Universal Robots URScript: screwdriver.script

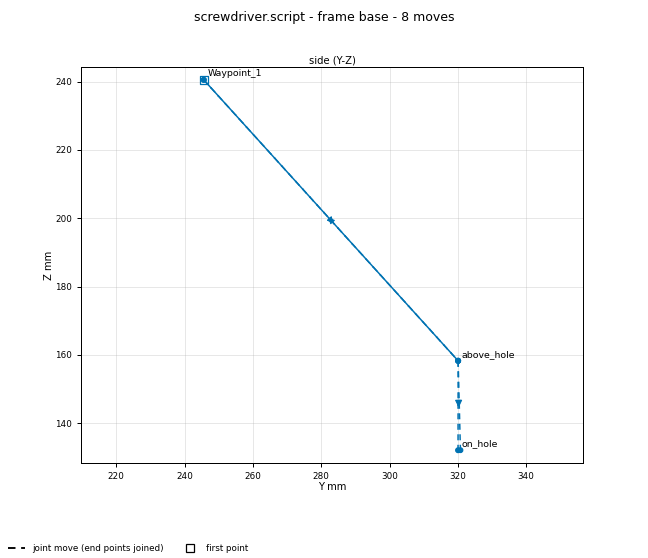
[picture p0: tool path of screwdriver.script in frame base, 8 of 54 moves have a stored position in this frame; points joined in program order, loops and branches not executed]
def unnamed():
  global _hidden_verificationVariable=0
  set_target_payload(1.710000, [0.052300, 0.000000, 0.046900], [0.000000, 0.000000, 0.000000, 0.000000, 0.000000, 0.000000])
  set_tool_communication(False, 115200, 0, 1, 1.5, 3.5)
  set_tool_output_mode(0)
  set_tool_digital_output_mode(0, 1)
  set_tool_digital_output_mode(1, 1)
  set_tool_voltage(0)
  set_gravity([0.0, 0.0, 9.82])
  set_safety_mode_transition_hardness(1)
  set_tcp(p[0.076,0.0,0.269,0.0,0.0,0.0])
  set_standard_analog_input_domain(0, 1)
  set_standard_analog_input_domain(1, 1)
  set_tool_analog_input_domain(0, 1)
  set_tool_analog_input_domain(1, 1)
  set_analog_outputdomain(0, 0)
  set_analog_outputdomain(1, 0)
  set_input_actions_to_default()
  global nb_vis_reusi=0
  global i_var_1=63
  global count_sec_touch=0
  global count_touch=0
  global erreur_vissage=0
  global perte_vis=0
  global count_vis=500
  global second_time_vis=0
  global rq_show_diag=0
  global count_pick_gig=5
  global count=495
  global should_i_vis=True
  # begin: URCap Installation Node
  #   Source: Robotiq_Screwdriving, 2.2.3.37910-alpha, Robotiq Inc.
  #   Type: Screwdriving
  #--------------------------------------------------------------------------------------------------
  # Screwdriver Constants
  #--------------------------------------------------------------------------------------------------
  RQ_REGULATION_MODE_CURRENT_WITH_RAMP_DOWN = 0
  RQ_REGULATION_MODE_ANGLE = 1
  RQ_REGULATION_MODE_TORQUE = 2
  RQ_REGULATION_MODE_SPEED = 3
  RQ_REGULATION_MODE_CURRENT = 4
  RQ_REGULATION_MODE_TIGHTENING = 5
  RQ_REGULATION_MODE_TORQUE_SPEED_CURRENT = 6
  RQ_ACTIVATE = True
  RQ_DIRECTION_CCW = False
  RQ_DIRECTION_CW = True
  RQ_MODE_NORMAL = False
  RQ_MODE_CALIBRATE = True
  RQ_SCREWDRIVER_ON = True
  RQ_SCREWDRIVER_OFF = False
  RQ_VACUUM_ON = True
  RQ_VACUUM_OFF = False
  RQ_MAX_SUPPLY_CURRENT_MA = 2000
  RQ_IN_ACTION = 0
  RQ_ANGLE_DETECTED = 1
  RQ_TORQUE_DETECTED = 2
  RQ_NO_DETECTION = 3
  RQ_SCREW_STATUS_ACTIVATION_IN_PROGRESS = 1
  RQ_SCREW_STATUS_ACTIVATION_DONE = 3
  RQ_SCREW_SUCCESS = 0
  RQ_SCREW_FAIL_ON_DISTANCE_MIN = 1
  RQ_SCREW_FAIL_ON_DISTANCE_MAX = 2
  RQ_SCREW_FAIL_ON_TIME_MAX = 3
  RQ_SCREW_FAIL_ON_SCREW_NOT_DETECTED = 4
  RQ_SCREW_FAIL_ON_SCREWDRIVER_NOT_ACTIVATED = 5
  RQ_SCREW_FAIL_ON_UNHANDLED_ERROR = 6
  RQ_SCREW_FAIL_ON_SCREWDRIVER_NOT_RESPONDING = 7
  RQ_SCREW_FAIL_ON_SCREWDRIVER_COMMUNICATION_LOST = 8
  RQ_SCREW_FAIL_ON_CONTACT_NOT_FOUND = 9
  RQ_SCREW_FAIL_WITHOUT_DETECTION = 10
  RQ_SCREW_SUCCESS_TEXT = "The screwdriving test is successful."
  RQ_SCREW_SUCCESS_TITLE_TEXT = "Screwdriving Test Success"
  RQ_PICK_SUCCESS = 0
  RQ_PICK_FAIL_ON_SCREW_NOT_READY = 1
  RQ_PICK_FAIL_ON_SCREW_NOT_DETECTED = 2
  RQ_PICK_FAIL_ON_FEEDER_NOT_READY = 3
  RQ_PICK_FAIL_ON_SCREWDRIVER_NOT_ACTIVATED = 5
  RQ_FEEDER_SCREW_PRESENT = 0
  RQ_PICK_SUCCESS_TEXT = "The pick test is successful."
  RQ_PICK_FAIL_ON_SCREW_NOT_READY_TEXT = "Screw not ready in feeder."
  RQ_PICK_FAIL_ON_SCREW_NOT_DETECTED_TEXT = "Screw not detected by screwdriver."
  RQ_PICK_FAIL_ON_FEEDER_NOT_READY_TEXT = "Feeder not ready."
  RQ_PICK_SUCCESS_TITLE_TEXT = "Pick Test Success"
  RQ_PICK_FAILED_TITLE_TEXT = "Pick Test Failed"
  RQ_SCREWDRIVER_NOT_ACTIVATED_TEXT = "Screwdriver is not activated. Please open Screwdriver Toolbar and click on Activate."
  RQ_MILLI_UNIT_TO_UNIT_FACTOR = 1000
  RQ_ENDLESS_TIMEOUT = 0
  RQ_UNUSED_PARAMETER = -1
  RQ_SCREW_FAIL_ON_DISTANCE_MIN_TEXT = "Minimum distance not reached."
  RQ_SCREW_FAIL_ON_DISTANCE_MAX_TEXT = "Maximum distance reached."
  RQ_SCREW_FAIL_ON_TIME_MAX_TEXT = "Maximum time reached."
  RQ_SCREW_FAIL_ON_NO_SCREW_TEXT = "No screw detected"
  RQ_SCREW_FAIL_TITLE = "Test Screw Failed"
  RQ_SCREW_FAIL_ON_UNHANDLED_ERROR_TEXT = "UE0 - Unhandled screw error"
  RQ_SCREW_FAIL_ON_SCREWDRIVER_NOT_RESPONDING_TEXT = "UE1 - Screwdriver not returning proper echo"
  RQ_SCREW_FAIL_ON_SCREWDRIVER_COMMUNICATION_LOST_TEXT = "UE2 - Screwdriver communication lost"
  RQ_SCREW_FAIL_ON_CONTACT_NOT_FOUND_TEXT = "UE3 - Contact with threads not found"
  RQ_SCREW_FAIL_WITHOUT_DETECTION_TEXT = "UE4 - Action finished without detection"
  RQ_TEACHING_OFF = 0
  RQ_TEACHING_ON = 1
  ###################################################
  #
  #  Fault types v2
  #
  ###################################################
  RQ_NO_FAULT = 0
  RQ_APPLICATION_WARNING = 1
  RQ_MOTOR_MINOR_ALARM = 2
  RQ_GENERAL_MINOR_ALARM = 4
  RQ_APPLICATION_MINOR_ALARM = 8
  RQ_MOTOR_MAJOR_ALARM = 16
  RQ_GENERAL_MAJOR_ALARM = 32
  RQ_APPLICATION_MAJOR_ALARM = 64
  RQ_CRITICAL_ALARM = 128

  RQ_NO_FAULT_MESSAGE = "NO_FAULT"
  RQ_APPLICATION_WARNING_MESSAGE = "APPLICATION_WARNING"
  RQ_MOTOR_MINOR_ALARM_MESSAGE = "MOTOR_MINOR_ALARM"
  RQ_GENERAL_MINOR_ALARM_MESSAGE = "GENERAL_MINOR_ALARM"
  RQ_APPLICATION_MINOR_ALARM_MESSAGE = "APPLICATION_MINOR_ALARM"
  RQ_MOTOR_MAJOR_ALARM_MESSAGE = "MOTOR_MAJOR_ALARM"
  RQ_GENERAL_MAJOR_ALARM_MESSAGE = "GENERAL_MAJOR_ALARM"
  RQ_APPLICATION_MAJOR_ALARM_MESSAGE = "APPLICATION_MAJOR_ALARM"
  RQ_CRITICAL_ALARM_MESSAGE = "CRITICAL_ALARM"

  ###################################################
  #
  #  Critical Alarm v2
  #
  ###################################################
  RQ_ACCELEROMETER_INIT = 1
  RQ_MOTOR_PWM_INIT = 2
  RQ_POSITION_SENSOR_INIT = 4
  RQ_GPIO_INIT = 8
  RQ_SOLENOID_INIT = 16
  RQ_FLASH_INIT = 32
  RQ_ADC_INIT = 64

  RQ_ACCELEROMETER_INIT_MESSAGE = "ACCELEROMETER_INIT"
  RQ_MOTOR_PWM_INIT_MESSAGE = "MOTOR_PWM_INIT"
  RQ_POSITION_SENSOR_INIT_MESSAGE = "POSITION_SENSOR_INIT"
  RQ_GPIO_INIT_MESSAGE = "GPIO_INIT"
  RQ_SOLENOID_INIT_MESSAGE = "SOLENOID_INIT"
  RQ_FLASH_INIT_MESSAGE = "FLASH_INIT"
  RQ_ADC_INIT_MESSAGE = "ADC_INIT"

  ###################################################
  #
  #  Application Warnings v2
  #
  ###################################################
  RQ_COMMUNICATION_NOT_READY = 1
  RQ_BLOCKED_AT_START = 2
  RQ_RESTRICTION_BEFORE_ANGLE = 4
  RQ_TIMEOUT = 8
  RQ_REG_WHILE_NOT_ACT = 16
  RQ_NOT_ACTIVATED = 32

  RQ_COMMUNICATION_NOT_READY_MESSAGE = "1 - COMMUNICATION_NOT_READY"
  RQ_BLOCKED_AT_START_MESSAGE = "2 - BLOCKED_AT_START"
  RQ_RESTRICTION_BEFORE_ANGLE_MESSAGE = "4 - RESTRICTION_BEFORE_ANGLE"
  RQ_TIMEOUT_MESSAGE = "8 - TIMEOUT"
  RQ_REGULATION_WHILE_NOT_ACT_MESSAGE = "16 - REGULATION_WHILE_NOT_ACT"
  RQ_NOT_ACTIVATED_MESSAGE = "32 - NOT_ACTIVATED"


  ###################################################
  #
  #  General Minor Alarm v2
  #
  ###################################################

  RQ_OVER_TEMPERATURE_SYSTEM = 2

  RQ_OVER_TEMPERATURE_SYSTEM_MESSAGE = "OVER_TEMPERATURE_SYSTEM"

  ###################################################
  #
  #  General Major Alarm v2
  #
  ###################################################

  RQ_E_STOP = 256
  RQ_OVER_CURRENT_SYSTEM = 512
  RQ_UNDER_VOLTAGE_24V = 1024
  RQ_UNDER_VOLTAGE_8V = 2048
  RQ_UNDER_VOLTAGE_3V = 4096

  RQ_E_STOP_MESSAGE = "E_STOP"
  RQ_OVER_CURRENT_SYSTEM_MESSAGE = "OVER_CURRENT_SYSTEM"
  RQ_UNDER_VOLTAGE_24V_MESSAGE = "UNDER_VOLTAGE_24V"
  RQ_UNDER_VOLTAGE_8V_MESSAGE = "UNDER_VOLTAGE_8V"
  RQ_UNDER_VOLTAGE_3V_MESSAGE = "UNDER_VOLTAGE_3V"

  ###################################################
  #
  #  Motor Minor Alarm v2
  #
  ###################################################
  RQ_CALIBRATION_PHASE_ERROR = 1
  RQ_CALIBRATION_POSITION_ERROR = 2
  RQ_CALIBRATION_PARAMETERS_ERROR = 4

  RQ_CALIBRATION_PHASE_ERROR_MESSAGE = "CALIBRATION_PHASE_ERROR"
  RQ_CALIBRATION_POSITION_ERROR_MESSAGE = "CALIBRATION_POSITION_ERROR"
  RQ_CALIBRATION_PARAMETERS_ERROR_MESSAGE = "CALIBRATION_PARAMETERS_ERROR"
  ###################################################
  #
  #  Motor Major Alarm v2
  #
  ###################################################
  RQ_UNDER_VOLTAGE = 1
  RQ_OVER_VOLTAGE = 2
  RQ_OVER_CURRENT_AC = 4
  RQ_OVER_CURRENT_DC = 8
  RQ_OVER_TEMP = 16
  RQ_POSITION_SENSOR_ERROR = 32
  RQ_PHASE_DRIVER_ERROR = 64
  RQ_PHASE_SENSOR_ERROR = 128

  RQ_UNDER_VOLTAGE_MESSAGE = "UNDER_VOLTAGE"
  RQ_OVER_VOLTAGE_MESSAGE = "OVER_VOLTAGE"
  RQ_OVER_CURRENT_AC_MESSAGE = "OVER_CURRENT_AC"
  RQ_OVER_CURRENT_DC_MESSAGE = "OVER_CURRENT_DC"
  RQ_OVER_TEMP_MESSAGE = "OVER_TEMP"
  RQ_POSITION_SENSOR_ERROR_MESSAGE = "POSITION_SENSOR_ERROR"
  RQ_PHASE_DRIVER_ERROR_MESSAGE = "PHASE_DRIVER_ERROR"
  RQ_PHASE_SENSOR_ERROR_MESSAGE = "PHASE_SENSOR_ERROR"
  global bash = rpc_factory("xmlrpc", "http://127.0.0.1:8000/bash")
  global logging_filename = str_cat("/tmp/screwing_info_",bash.date("+%Y_%m_%d_%H:%M:%S.csv"))
  #--------------------------------------------------------------------------------------------------
  #   Faults               2000[7-0]   Screwdriver fault types:
  #                                   0 = application warnings.[2501]
  #                                   1 = motor minor[2505]
  #                                   2 = general minor[2504]
  #                                   3 = application minor[2502]
  #                                   4 = motor major[2506]
  #                                   5 = general major[2504]
  #                                   6 = application major[2503]
  #                                   7 = critical[2500]
  #--------------------------------------------------------------------------------------------------
  def rq_get_screw_fault(slave_id=9):
    rq_error_list = [0,0,0,0,0,0,0,0]
    registers_200x = rq_comm_read_registers_200x(slave_id, RQ_READ_SCREWDRIVER_REGISTERS_SIZE)
    rq_error_type = registers_200x[0]

    if (rq_error_type == RQ_NO_FAULT):
      return rq_error_list
    end

    registers_250x = rq_comm_read_registers_250x(slave_id)
    rq_application_warnings = rq_extract_boolean_from_register_value(rq_error_type, 0)
    rq_motor_minor = rq_extract_boolean_from_register_value(rq_error_type, 1)
    rq_general_minor = rq_extract_boolean_from_register_value(rq_error_type, 2)
    rq_application_minor = rq_extract_boolean_from_register_value(rq_error_type, 3)
    rq_motor_major = rq_extract_boolean_from_register_value(rq_error_type, 4)
    rq_general_major = rq_extract_boolean_from_register_value(rq_error_type, 5)
    rq_application_major = rq_extract_boolean_from_register_value(rq_error_type, 6)
    rq_critical = rq_extract_boolean_from_register_value(rq_error_type, 7)

    if(rq_application_warnings):
     rq_error_list[0] = rq_extract_value_from_register_value(registers_250x[1], 0, 16)
    end
    if(rq_motor_minor):
     rq_error_list[1] = rq_extract_value_from_register_value(registers_250x[5], 0, 16)
    end
    if(rq_general_minor):
     rq_error_list[2] = rq_extract_value_from_register_value(registers_250x[4], 0, 8)
    end
    if(rq_application_minor):
     rq_error_list[3] = rq_extract_value_from_register_value(registers_250x[2], 0, 16)
    end
    if(rq_motor_major):
     rq_error_list[4] = rq_extract_value_from_register_value(registers_250x[6], 0, 16)
    end
    if(rq_general_major):
     rq_error_list[5] = rq_extract_value_from_register_value(registers_250x[4], 8, 16)
    end
    if(rq_application_major):
     rq_error_list[6] = rq_extract_value_from_register_value(registers_250x[3], 0, 16)
    end
    if(rq_critical):
     rq_error_list[7] = rq_extract_value_from_register_value(registers_250x[0], 0, 16)
    end

    return rq_error_list
  end

  #--------------------------------------------------------------------------------------------------
  #   Activate echo       2000[8]     Echo of the activate
  #--------------------------------------------------------------------------------------------------
  def rq_get_screw_activated_echo(slave_id=9):
      registers_200x = rq_comm_read_registers_200x(slave_id, RQ_READ_SCREWDRIVER_REGISTERS_SIZE)
      return rq_extract_is_screw_activated_echo(registers_200x)
  end
  def rq_extract_is_screw_activated_echo(registers_200x):
      return rq_extract_boolean_from_register_value(registers_200x[0], 8)
  end

  def rq_get_activation_and_screw_detection(slave_id):
    registers_200x = rq_comm_read_registers_200x(slave_id, RQ_READ_SCREWDRIVER_REGISTERS_SIZE)
    activation = rq_extract_is_screw_activated_echo(registers_200x)
    screw_detection = rq_extract_boolean_from_register_value(registers_200x[1], 12)

    return [activation, screw_detection]
  end
  #--------------------------------------------------------------------------------------------------
  #   Direction echo      2000[9]     Echo of the desired direction.
  #--------------------------------------------------------------------------------------------------
  def rq_get_screw_direction_echo(slave_id=9):
      registers_200x = rq_comm_read_registers_200x(slave_id, RQ_READ_SCREWDRIVER_REGISTERS_SIZE)
      return rq_extract_screw_direction_echo(registers_200x)
  end
  def rq_extract_screw_direction_echo(registers_200x):
      return rq_extract_boolean_from_register_value(registers_200x[0], 9)
  end

  #--------------------------------------------------------------------------------------------------
  #   Regulate echo       2000[11]    Echo of the regulate.
  #--------------------------------------------------------------------------------------------------
  def rq_get_screw_regulate_echo(slave_id=9):
      registers_200x = rq_comm_read_registers_200x(slave_id, RQ_READ_SCREWDRIVER_REGISTERS_SIZE)
      return rq_extract_screw_regulate_echo(registers_200x)
  end
  def rq_extract_screw_regulate_echo(registers_200x):
      return rq_extract_boolean_from_register_value(registers_200x[0], 11)
  end

  #--------------------------------------------------------------------------------------------------
  #   Screwdriver status  2000[13-12]     3 = Activation done
  #                                       1 = Activation in progress
  #                                       0 = Else
  #--------------------------------------------------------------------------------------------------
  def rq_get_screw_status(slave_id=9):
      registers_200x = rq_comm_read_registers_200x(slave_id, RQ_READ_SCREWDRIVER_REGISTERS_SIZE)
      return rq_extract_screw_status_echo(registers_200x)
  end
  def rq_extract_screw_status_echo(registers_200x):
      return rq_extract_value_from_register_value(registers_200x[0], 12, 2)
  end
  #--------------------------------------------------------------------------------------------------
  #   Action status       2000[15-14]     0 = initiating/doing an action
  #                                       1 = angle detected
  #                                       2 = torque detected
  #                                       3 = action finished without detection
  #--------------------------------------------------------------------------------------------------
  def rq_get_screw_action(slave_id=9):
      registers_200x = rq_comm_read_registers_200x(slave_id, RQ_READ_SCREWDRIVER_REGISTERS_SIZE)
      return rq_extract_value_from_register_value(registers_200x[0], 14, 2)
  end

  #--------------------------------------------------------------------------------------------------
  #   Regulation mode echo   2001[2-0]    0 = regulates speed, stops at desired current or timeout (ramp down at angle)
  #                                       1 = regulates speed, stops at desired current or timeout
  #                                       2 = regulates speed, stops at desired angle or timeout
  #                                       3 = regulates current, stops at timeout
  #                                       4 = regulates speed, stops at timeout
  #                                       5 = ?
  #                                       6 = regulate torque at stall (internal mode)
  #                                       7 = regultate torque (internal mode)
  #--------------------------------------------------------------------------------------------------
  def rq_get_screw_regulation_mode_echo(slave_id=9):
      registers_200x = rq_comm_read_registers_200x(slave_id, RQ_READ_SCREWDRIVER_REGISTERS_SIZE)
      return rq_extract_regulation_mode_echo(registers_200x)
  end
  def rq_extract_regulation_mode_echo(registers_200x):
      return rq_extract_value_from_register_value(registers_200x[1], 0, 2)
  end

  #--------------------------------------------------------------------------------------------------
  #   Vacuum screw detection 2001[12]     0 = not detected
  #                                       1 = detected
  #--------------------------------------------------------------------------------------------------
  def rq_is_screw_detected(slave_id=9):
      registers_200x = rq_comm_read_registers_200x(slave_id, RQ_READ_SCREWDRIVER_REGISTERS_SIZE)
      return rq_extract_boolean_from_register_value(registers_200x[1], 12)
  end

  #--------------------------------------------------------------------------------------------------
  #   Vacuum echo            2001[13]     0 = close
  #                                       1 = open
  #--------------------------------------------------------------------------------------------------
  def rq_get_screw_vacuum_echo(slave_id=9):
      registers_200x = rq_comm_read_registers_200x(slave_id, RQ_READ_SCREWDRIVER_REGISTERS_SIZE)
      return rq_extract_screw_vacuum_echo(registers_200x)
  end
  def rq_extract_screw_vacuum_echo(registers_200x):
      return rq_extract_boolean_from_register_value(registers_200x[1], 13)
  end

  #--------------------------------------------------------------------------------------------------
  #   Operation mode echo    2001[14]    Echo of the screwdriver mode
  #--------------------------------------------------------------------------------------------------
  def rq_get_screw_operation_mode_echo(slave_id=9):
      registers_200x = rq_comm_read_registers_200x(slave_id, RQ_READ_SCREWDRIVER_REGISTERS_SIZE)
      return rq_extract_screw_operation_mode(registers_200x)
  end
  def rq_extract_screw_operation_mode(registers_200x):
      return rq_extract_boolean_from_register_value(registers_200x[1], 14)
  end

  #--------------------------------------------------------------------------------------------------
  #   Rotation current echo   2002        Desired current to apply. 1 bit = 1 mA
  #--------------------------------------------------------------------------------------------------
  def rq_get_screw_rotation_current_echo_mA(slave_id=9):
      registers_200x = rq_comm_read_registers_200x(slave_id, RQ_READ_SCREWDRIVER_REGISTERS_SIZE)
      return rq_extract_rotation_current_echo(registers_200x)
  end
  def rq_extract_rotation_current_echo(registers_200x):
      return registers_200x[2]
  end

  #--------------------------------------------------------------------------------------------------
  #   Rotation speed echo     2003        Desired rotation speed to regulate in RPM
  #--------------------------------------------------------------------------------------------------
  def rq_get_screw_rotation_speed_echo_rpm(slave_id=9):
      registers_200x = rq_comm_read_registers_200x(slave_id, RQ_READ_SCREWDRIVER_REGISTERS_SIZE)
      return rq_extract_screw_rotation_speed_echo_rpm(registers_200x)
  end
  def rq_extract_screw_rotation_speed_echo_rpm(registers_200x):
      return registers_200x[3]
  end

  #--------------------------------------------------------------------------------------------------
  #   Actual delta angle      2004[15-0]-2005[15-8]    Actual delta angle in degrees
  #--------------------------------------------------------------------------------------------------
  def rq_get_screw_delta_angle_deg(slave_id=9):
      registers_200x = rq_comm_read_registers_200x(slave_id, RQ_READ_SCREWDRIVER_REGISTERS_SIZE)
      register_2005_8_15 = rq_extract_value_from_register_value(registers_200x[5], 8, 8)
      return registers_200x[4] + register_2005_8_15 * pow(2, 16)
  end

  #--------------------------------------------------------------------------------------------------
  #   Desired delta angle      2007[15-0]-2008[15-8]    Desired delta angle in degrees
  #--------------------------------------------------------------------------------------------------
  def rq_get_desired_delta_angle_deg(slave_id=9):
      registers_200x = rq_comm_read_registers_200x(slave_id, RQ_READ_SCREWDRIVER_REGISTERS_SIZE)
      register_2008_8_15 = rq_extract_value_from_register_value(registers_200x[8], 8, 8)
      return registers_200x[7] + register_2008_8_15 * pow(2, 16)
  end

  #--------------------------------------------------------------------------------------------------
  #   Actual current          2005[7-0]  Actual current, 1 bit = 100 mA
  #--------------------------------------------------------------------------------------------------
  def rq_get_screw_current_mA(slave_id=9):
      registers_200x = rq_comm_read_registers_200x(slave_id, RQ_READ_SCREWDRIVER_REGISTERS_SIZE)
      register_2005_0_7 = rq_extract_value_from_register_value(registers_200x[5], 0, 8)
      return register_2005_0_7 * 100
  end

  #--------------------------------------------------------------------------------------------------
  #   Actual rotation speed   2006    Actual rotation speed   RPM
  #--------------------------------------------------------------------------------------------------
  def rq_get_screw_rotation_speed_rpm(slave_id=9):
      registers_200x = rq_comm_read_registers_200x(slave_id, RQ_READ_SCREWDRIVER_REGISTERS_SIZE)
      return registers_200x[6]
  end

  #--------------------------------------------------------------------------------------------------
  #   Torque Threshold        2010
  #--------------------------------------------------------------------------------------------------
  def rq_get_torque_threshold_Nm(slave_id=9):
      registers_200x = rq_comm_read_registers_200x(slave_id, RQ_READ_SCREWDRIVER_REGISTERS_SIZE)
      return rq_extract_torque_threshold_echo(registers_200x) / 10000
  end
  def rq_extract_torque_threshold_echo(registers_200x):
      return rq_convert_unsigned16_to_signed16(registers_200x[10])
  end

  #--------------------------------------------------------------------------------------------------
  #   Torque Angle Slope      2011
  #--------------------------------------------------------------------------------------------------
  def rq_get_torque_slope(slave_id=9):
      registers_200x = rq_comm_read_registers_200x(slave_id, RQ_READ_SCREWDRIVER_REGISTERS_SIZE)
      return rq_extract_torque_angle_slope_echo(registers_200x)
  end
  def rq_extract_torque_angle_slope_echo(registers_200x):
      return rq_convert_unsigned16_to_signed16(registers_200x[11])
  end

  #--------------------------------------------------------------------------------------------------
  #   Torque Gain %     2012  value between 0 and 100. Default is 12
  #--------------------------------------------------------------------------------------------------
  def rq_get_torque_gain_pct(slave_id=9):
      registers = rq_read_registers(slave_id, 2012, 1, rq_xml_rpc_modbus_debug)
      return registers[0]
  end

  #--------------------------------------------------------------------------------------------------
  #   Debug register          6021
  #--------------------------------------------------------------------------------------------------
  def rq_get_screw_register_6021(slave_id=9):
      register_6020 = rq_comm_read_3_registers_6020(slave_id)

      return register_6020[1]
  end

  #--------------------------------------------------------------------------------------------------
  #   Debug register          6022
  #--------------------------------------------------------------------------------------------------
  def rq_get_screw_register_6022(slave_id=9):
      register_6020 = rq_comm_read_3_registers_6020(slave_id)

      return register_6020[2]
  end

  #--------------------------------------------------------------------------------------------------
  # Look for screwdriver activation
  #--------------------------------------------------------------------------------------------------
  def rq_screwdriver_is_activated(slave_id=9):
    registers_200x = rq_comm_read_registers_200x(slave_id, RQ_READ_SCREWDRIVER_REGISTERS_SIZE)

    return (rq_extract_screw_status_echo(registers_200x) == RQ_SCREW_STATUS_ACTIVATION_DONE) and rq_extract_is_screw_activated_echo(registers_200x)
  end

  #--------------------------------------------------------------------------------------------------
  # Returns True when all echo matches parameters
  #--------------------------------------------------------------------------------------------------
  def rq_screwdriver_echo_equal(slave_id, vacuum, rotation_current, regulate, direction, rotation_speed, operation_mode, regulation_mode, torque_threshold, torque_angle_slope):
    registers_200x = rq_comm_read_registers_200x(slave_id, RQ_READ_SCREWDRIVER_REGISTERS_SIZE)

    return (vacuum == rq_extract_screw_vacuum_echo(registers_200x)) and
           (rotation_current == rq_extract_rotation_current_echo(registers_200x)) and
           (regulate == rq_extract_screw_regulate_echo(registers_200x)) and
           (direction == rq_extract_screw_direction_echo(registers_200x)) and
           (rotation_speed == rq_extract_screw_rotation_speed_echo_rpm(registers_200x)) and
           (operation_mode == rq_extract_screw_operation_mode(registers_200x)) and
           (regulation_mode == rq_extract_regulation_mode_echo(registers_200x)) and
           (torque_threshold == rq_extract_torque_threshold_echo(registers_200x)) and
           (torque_angle_slope == rq_extract_torque_angle_slope_echo(registers_200x))

  end

  #--------------------------------------------------------------------------------------------------
  # Refresh registers 200x to get actual communication state. Return communication state.
  #--------------------------------------------------------------------------------------------------
  def rq_is_comm_lost(slave_id):
    rq_comm_read_registers_200x(slave_id, RQ_READ_SCREWDRIVER_REGISTERS_SIZE)

    return rq_comm_lost[rq_comm_slave_id_to_index(slave_id)]
  end

  #--------------------------------------------------------------------------------------------------
  # Returns the magnetic encoder count - Register 4000(LSB) - 4001(MSB)
  #--------------------------------------------------------------------------------------------------
  def rq_get_magnetic_encoder_count(slave_id=9):
      registers_lsb = rq_read_registers(slave_id, 4000, 1, rq_xml_rpc_modbus_debug)
      registers_msb = rq_read_registers(slave_id, 4001, 1, rq_xml_rpc_modbus_debug)

      return (registers_msb[0] * pow(2,16)) + registers_lsb[0]
  end

  #--------------------------------------------------------------------------------------------------
  # Returns the magnetic encoder error flag - Register 4002[15-13]
  #                                                         13 = Framing error
  #                                                         14 = Invalid command error
  #                                                         15 = Parity error
  #--------------------------------------------------------------------------------------------------
  def rq_get_magnetic_encoder_error_flag(slave_id=9):
      registers = rq_read_registers(slave_id, 4002, 1, rq_xml_rpc_modbus_debug)

      if (rq_extract_boolean_from_register_value(registers[0], 13)):
        return "Encoder error - Framing error"
      elif (rq_extract_boolean_from_register_value(registers[0], 14)):
        return "Encoder error - Invalid command error"
      elif (rq_extract_boolean_from_register_value(registers[0], 15)):
        return "Encoder error - Parity error"
      end

      return "No magnetic encoder error"
  end

  #--------------------------------------------------------------------------------------------------
  # Returns the magnetic encoder is ready - Register 4002[8]
  #--------------------------------------------------------------------------------------------------
  def rq_get_magnetic_encoder_ready(slave_id=9):
      registers = rq_read_registers(slave_id, 4002, 1,rq_xml_rpc_modbus_debug)

      return not rq_extract_boolean_from_register_value(registers[0], 8)
  end

  #--------------------------------------------------------------------------------------------------
  # Returns the magnetic encoder field strength - Register 4002[7-0]
  #--------------------------------------------------------------------------------------------------
  def rq_get_magnetic_encoder_field_strength(slave_id=9):
      registers = rq_read_registers(slave_id, 4002, 1, rq_xml_rpc_modbus_debug)

      return rq_extract_value_from_register_value(registers[0], 0, 8)
  end

  #--------------------------------------------------------------------------------------------------
  # Returns the CPU percent max live - Register 4003
  #--------------------------------------------------------------------------------------------------
  def rq_get_cpu_percent_max_live(slave_id=9):
      registers = rq_read_registers(slave_id, 4003, 1,rq_xml_rpc_modbus_debug)

      return registers[0]
  end

  #--------------------------------------------------------------------------------------------------
  # Returns the CPU percent max since boot - Register 4004
  #--------------------------------------------------------------------------------------------------
  def rq_get_cpu_percent_max_since_boot(slave_id=9):
      registers = rq_read_registers(slave_id, 4004, 1, rq_xml_rpc_modbus_debug)

      return registers[0]
  end

  #--------------------------------------------------------------------------------------------------
  # Returns the current motor analog Amps - Register 4005
  #--------------------------------------------------------------------------------------------------
  def rq_get_current_motor_amps(slave_id=9):
      registers = rq_read_registers(slave_id, 4005, 1, rq_xml_rpc_modbus_debug)

      return registers[0]/100
  end

  #--------------------------------------------------------------------------------------------------
  # Returns the analog 24v voltage - Register 4006
  #--------------------------------------------------------------------------------------------------
  def rq_get_analog_24_volt(slave_id=9):
      registers =rq_read_registers(slave_id, 4006, 1, rq_xml_rpc_modbus_debug)

      return registers[0]/100
  end

  #--------------------------------------------------------------------------------------------------
  # Returns the analog 8v8 voltage - Register 4007
  #--------------------------------------------------------------------------------------------------
  def rq_get_analog_8v8_volt(slave_id=9):
      registers = rq_read_registers(slave_id, 4007, 1, rq_xml_rpc_modbus_debug)

      return registers[0]/100
  end

  #--------------------------------------------------------------------------------------------------
  # Returns the microcontroller temperature Celsius - Register 4008
  #--------------------------------------------------------------------------------------------------
  def rq_get_uc_temp_celsius(slave_id=9):
      registers = rq_read_registers(slave_id, 4008, 1, rq_xml_rpc_modbus_debug)

      return registers[0]/100
  end

  #--------------------------------------------------------------------------------------------------
  # Returns the motor temperature Celsius - Register 4009
  #--------------------------------------------------------------------------------------------------
  def rq_get_motor_temp_celsius(slave_id=9):
      registers = rq_read_registers(slave_id, 4009, 1,rq_xml_rpc_modbus_debug)

      return registers[0]/100
  end

  #--------------------------------------------------------------------------------------------------
  # Returns the vacuum pressure Psi - Register 4010
  #--------------------------------------------------------------------------------------------------
  def rq_get_vacuum_pressure_kpa(slave_id=9):
      registers = rq_read_registers(slave_id, 4010, 1, rq_xml_rpc_modbus_debug)

      return rq_convert_unsigned16_to_signed16(registers[0]) / 100
  end

  #--------------------------------------------------------------------------------------------------
  # Returns the estimated load torque - Register 4012
  #--------------------------------------------------------------------------------------------------
  def rq_get_load_nm(slave_id=9):
      registers = rq_read_registers(slave_id, 4012, 1, rq_xml_rpc_modbus_debug)

      return registers[0]/1000
  end

  #--------------------------------------------------------------------------------------------------
  # Returns the estimated maximum load torque - Register 4013
  #--------------------------------------------------------------------------------------------------
  def rq_get_max_load_nm(slave_id=9):
      registers = rq_read_registers(slave_id, 4013, 1, rq_xml_rpc_modbus_debug)

      return registers[0]/1000
  end

  #--------------------------------------------------------------------------------------------------
  # add all diagnostic registers output in Polyscope Log tab.
  #--------------------------------------------------------------------------------------------------
  def rq_log_screw_diag_registers(slave_id=9):
    textmsg("magnetic encoder count : ", rq_get_magnetic_encoder_count(slave_id))
    textmsg("magnetic encoder is ready : ", rq_get_magnetic_encoder_ready(slave_id))
    textmsg("magnetic encoder error flag : ", rq_get_magnetic_encoder_error_flag(slave_id))
    textmsg("magnetic encoder field strength : ", rq_get_magnetic_encoder_field_strength(slave_id))
    textmsg("CPU percent max LIVE : ", rq_get_cpu_percent_max_live(slave_id))
    textmsg("CPU percent max since boot : ", rq_get_cpu_percent_max_since_boot(slave_id))
    textmsg("current motor analog Amps : ", rq_get_current_motor_amps(slave_id))
    textmsg("analog 24v voltage : ", rq_get_analog_24_volt(slave_id))
    textmsg("analog 8v8 voltage : ", rq_get_analog_8v8_volt(slave_id))
    textmsg("microcontroller temp Celsius : ", rq_get_uc_temp_celsius(slave_id))
    textmsg("motor temp Celsius : ", rq_get_motor_temp_celsius(slave_id))
    textmsg("vacuum pressure Kpa : ", rq_get_vacuum_pressure_kpa(slave_id))
    textmsg("estimated load torque Nm LIVE : ", rq_get_load_nm(slave_id))
    textmsg("estimated maximum load torque Nm :", rq_get_max_load_nm(slave_id))
  end

  #--------------------------------------------------------------------------------------------------
  #   Pressure sensor offset        441 (100bit = kPa (signed))
  #                                 pressure_offset in kpa
  #
  #--------------------------------------------------------------------------------------------------
  def get_pressure_sensor_offset(slave_id = 9):
    registers = rq_read_registers(slave_id, 441, 1, rq_xml_rpc_modbus_debug)

    return rq_convert_unsigned16_to_signed16(registers[0]) / 100
  end

  #--------------------------------------------------------------------------------------------------
  # Convert unsigned 16 bits integer to signed 16 bits integer
  #--------------------------------------------------------------------------------------------------
  def rq_convert_unsigned16_to_signed16(value):
    if (value >= 32768):
      return value - 65536
    end
    return value
  end
  #--------------------------------------------------------------------------------------------------
  #   Register            1000        Action request
  #
  #   Regulation mode     1000[2-0]   0 = regulates speed, stops at desired current or timeout
  #                                   1 = regulates speed, with ramp down, stops at desired angle or timeout
  #                                   2-7 = unused
  #   Activate            1000[8]     0 = Resetting errors
  #                                   1 = Allows the screwdriver to do an action
  #   Rotation direction  1000[9]     0 = Clockwise (screwing)
  #                                   1 = Counter-clockwise (unscrewing)
  #   Regulate            1000[11]    0 = doing nothing (stop movement)
  #                                   1 = regulating movement
  #   Teaching            1000[12]    0 = inactive
  #                                   1 = active
  #   Vacuum activation   1000[13]    0 = close
  #                                   1 = open
  #   Operation mode      1000[14]    0 = normal mode (Torque mode)
  #                                   1 = calibration mode (Current Mode)
  #   Command modify      1000[15]    0 = new command
  #                                   1 = modify command
  #--------------------------------------------------------------------------------------------------
  #   Register            1001[15-0]  Max supply current
  #                                   Range 0-65535 (1 bit = 1 mA)
  #--------------------------------------------------------------------------------------------------
  #   Register            1002[15-0]   Desired rotation current
  #                                    Range 0-65535 (1 bit = 1 mA)
  #--------------------------------------------------------------------------------------------------
  #   Register            1003        Desired rotation speed in RPM
  #                                   Range 16bit = 65Krpm
  #--------------------------------------------------------------------------------------------------
  #   Register            1004[15-0]-1005[15-8]   Desired rotation delta angle
  #                                               Desired delta angle to attain
  #                                               24bit = 46 kdegrees
  #--------------------------------------------------------------------------------------------------
  #   Register            1005[7-0]   Rotation timeout
  #                                   Timeout of regulated movement (8bit = 25.5s), 1bit = 0.1s
  #--------------------------------------------------------------------------------------------------
  #   Register            1006        Torque Threshold
  #
  #--------------------------------------------------------------------------------------------------
  #   Register            1007        Torque Angle Slope
  #
  #--------------------------------------------------------------------------------------------------
  def rq_set_screw_registers_100x(slave_id, regulation_mode, activate, direction, operation_mode, regulate, teaching,
  vacuum, rotation_current, max_supply_current_mA, rotation_speed_rpm, rotation_delta_angle, rotation_timeout_ms,
  torque_threshold, torque_angle_slope, modify_command = False):
      registers_100x = [0, 0, 0, 0, 0, 0, 0, 0]
      registers_100x[0] = rq_insert_value_in_register_value(registers_100x[0], 0, 3, regulation_mode)
      registers_100x[0] = rq_insert_boolean_in_register_value(registers_100x[0], 8, activate)
      registers_100x[0] = rq_insert_boolean_in_register_value(registers_100x[0], 9, direction)
      registers_100x[0] = rq_insert_boolean_in_register_value(registers_100x[0], 11, regulate)
      registers_100x[0] = rq_insert_value_in_register_value(registers_100x[0], 12, 1, teaching)
      registers_100x[0] = rq_insert_boolean_in_register_value(registers_100x[0], 13, vacuum)
      registers_100x[0] = rq_insert_boolean_in_register_value(registers_100x[0], 14, operation_mode)
      registers_100x[0] = rq_insert_boolean_in_register_value(registers_100x[0], 15, modify_command)

      registers_100x[1] = max_supply_current_mA

      registers_100x[2] = rotation_current

      registers_100x[3] = rotation_speed_rpm

      rotation_angle_lsb = floor(rotation_delta_angle % pow(2, 16))
      rotation_angle_msb = floor((rotation_delta_angle -  rotation_angle_lsb) / pow(2, 16))

      registers_100x[4] = rotation_angle_lsb
      registers_100x[5] = rq_insert_msb_in_register_value(registers_100x[5], rotation_angle_msb)
      registers_100x[5] = rq_insert_lsb_in_register_value(registers_100x[5], floor(rotation_timeout_ms / 100))

      registers_100x[6] = torque_threshold
      registers_100x[7] = torque_angle_slope

      rq_comm_write_registers_100x(slave_id, registers_100x, 8)
  end

  #--------------------------------------------------------------------------------------------------
  #   Activate screwdriver, sequence:
  #   1 - Reset screwdriver (activate = False) and wait echo
  #   2 - Activate screwdriver (activate = True) and wait echo and status
  #--------------------------------------------------------------------------------------------------
  def rq_screw_activate(slave_id = 9):
      while(rq_get_screw_activated_echo(slave_id)):
          registers_100x = rq_comm_get_registers_100x(slave_id, 8)
          registers_100x[0] = rq_insert_boolean_in_register_value(registers_100x[0], 8, False)
          rq_comm_write_registers_100x(slave_id, registers_100x, 8)
          sleep(0.1)
      end

      while(not rq_get_screw_activated_echo(slave_id) or rq_get_screw_status(slave_id) != RQ_SCREW_STATUS_ACTIVATION_DONE):
          registers_100x = rq_comm_get_registers_100x(slave_id, 8)
          registers_100x[0] = rq_insert_boolean_in_register_value(registers_100x[0], 8, True)
          rq_comm_write_registers_100x(slave_id, registers_100x, 8)
          sleep(0.1)
      end
  end

  #--------------------------------------------------------------------------------------------------
  #   Regulate            1000[11]    0 = doing nothing (stop movement)
  #                                   1 = regulating movement
  #--------------------------------------------------------------------------------------------------
  def rq_set_screw_regulate(slave_id, regulate):
      registers_100x = rq_comm_get_registers_100x(slave_id, 8)
      registers_100x[0] = rq_insert_boolean_in_register_value(registers_100x[0], 11, regulate)
      rq_comm_write_registers_100x(slave_id, registers_100x, 8)
  end

  #--------------------------------------------------------------------------------------------------
  #   Torque gain %            1008   torque gain is a value between 0 and 100. The default value is 12.
  #
  #--------------------------------------------------------------------------------------------------
  def rq_set_torque_gain_pct(torque_gain = 12, slave_id=9):
    rq_write_registers(slave_id, 1008, [torque_gain], rq_xml_rpc_modbus_debug)
  end

  #--------------------------------------------------------------------------------------------------
  #   Vacuum command on
  #--------------------------------------------------------------------------------------------------
  def rq_screw_vacuum_on(slave_id = 9):
      rq_set_screw_vacuum(True, slave_id)
  end

  #--------------------------------------------------------------------------------------------------
  #   Vacuum command off
  #--------------------------------------------------------------------------------------------------
  def rq_screw_vacuum_off(slave_id = 9):
      rq_set_screw_vacuum(False, slave_id)
  end

  #--------------------------------------------------------------------------------------------------
  #   Vacuum command off and regulate to false
  #--------------------------------------------------------------------------------------------------

  def rq_screw_vacuum_off_and_stop_regulate(slave_id=9):
    registers_100x = rq_comm_get_registers_100x(slave_id, 8)
    registers_200x = rq_comm_read_registers_200x(slave_id, RQ_READ_SCREWDRIVER_REGISTERS_SIZE)

    activate = rq_extract_boolean_from_register_value(registers_200x[0], 8)
    rotation_direction = rq_extract_boolean_from_register_value(registers_200x[0], 9)
    regulation_mode = rq_extract_value_from_register_value(registers_200x[1], 0, 2)
    operation_mode = rq_extract_value_from_register_value(registers_200x[1], 14, 1)
    regulate = False
    vacuum = False

    registers_100x[0] = rq_insert_value_in_register_value(registers_100x[0], 0, 2, regulation_mode)
    registers_100x[0] = rq_insert_boolean_in_register_value(registers_100x[0], 8, activate)
    registers_100x[0] = rq_insert_boolean_in_register_value(registers_100x[0], 9, rotation_direction)
    registers_100x[0] = rq_insert_boolean_in_register_value(registers_100x[0], 11, regulate)
    registers_100x[0] = rq_insert_boolean_in_register_value(registers_100x[0], 13, vacuum)
    registers_100x[0] = rq_insert_value_in_register_value(registers_100x[0], 14, 2, operation_mode)

    rq_comm_write_registers_100x(slave_id, registers_100x, 8)
  end

  #--------------------------------------------------------------------------------------------------
  #   Vacuum command         1000[13]     0 = close
  #                                       1 = open
  #--------------------------------------------------------------------------------------------------
  def rq_set_screw_vacuum(vacuum, slave_id = 9):
    registers_100x = rq_comm_get_registers_100x(slave_id, 8)
    registers_200x = rq_comm_read_registers_200x(slave_id, RQ_READ_SCREWDRIVER_REGISTERS_SIZE)

    activate = rq_extract_boolean_from_register_value(registers_200x[0], 8)
    rotation_direction = rq_extract_boolean_from_register_value(registers_200x[0], 9)
    regulate = rq_extract_boolean_from_register_value(registers_200x[0], 11)
    regulation_mode = rq_extract_value_from_register_value(registers_200x[1], 0, 2)
    operation_mode = rq_extract_value_from_register_value(registers_200x[1], 14, 1)

    registers_100x[0] = rq_insert_value_in_register_value(registers_100x[0], 0, 2, regulation_mode)
    registers_100x[0] = rq_insert_boolean_in_register_value(registers_100x[0], 8, activate)
    registers_100x[0] = rq_insert_boolean_in_register_value(registers_100x[0], 9, rotation_direction)
    registers_100x[0] = rq_insert_boolean_in_register_value(registers_100x[0], 11, regulate)
    registers_100x[0] = rq_insert_boolean_in_register_value(registers_100x[0], 13, vacuum)
    registers_100x[0] = rq_insert_value_in_register_value(registers_100x[0], 14, 2, operation_mode)

    rq_comm_write_registers_100x(slave_id, registers_100x, 8)
  end

  #--------------------------------------------------------------------------------------------------
  #   Set Pressure sensor offset        441 (100bit = kPa (signed))
  #                                      pressure_offset in kpa
  #
  #--------------------------------------------------------------------------------------------------
  def set_pressure_sensor_offset(pressure_offset=0, slave_id = 9):
    SAVE_PRESSURE_OFFSET = 56
    KPA_TO_BIT = 100

    offset_in_bit = rq_convert_unsigned32_to_signed16(pressure_offset * KPA_TO_BIT)
    rq_write_registers(slave_id, 441, [offset_in_bit], rq_xml_rpc_modbus_debug)

    save_pressure_offset_msb = floor(SAVE_PRESSURE_OFFSET * pow(2,8))
    rq_write_registers(slave_id, 440, [save_pressure_offset_msb], rq_xml_rpc_modbus_debug)
  end

  #--------------------------------------------------------------------------------------------------
  # Convert unsigned 32 bits integer to signed 16 bits integer
  #--------------------------------------------------------------------------------------------------
  def rq_convert_unsigned32_to_signed16(value):
    if (value < 0):
      return value + 65536
    end
    return value
  end

  #--------------------------------------------------------------------------------------------------
  #   Reset Pressure sensor offset to ambient pressure       440
  #
  #--------------------------------------------------------------------------------------------------
  def reset_pressure_sensor_offset(slave_id = 9):
    RESET_PRESSURE_OFFSET = 131

    reset_pressure_offset_msb = floor(RESET_PRESSURE_OFFSET * pow(2,8))
    rq_write_registers(slave_id, 440, [reset_pressure_offset_msb], rq_xml_rpc_modbus_debug)
  end
  global rq_feeder_timeout = 90
  global rq_pick_rotation_speed = 200

  def rq_is_feeder_screw_ready(ready_input):
    return get_standard_digital_in(ready_input)
  end

  def rq_is_feeder_status_ok(feeder_status):
    return get_standard_digital_in(feeder_status)
  end

  def rq_wait_for_feeder_status_ok(feeder_status, timeout):
    time_step = 0.008

    if(not rq_is_feeder_status_ok(feeder_status)):
      textmsg("Waiting for feeder status.")
    end

    while((not rq_is_feeder_status_ok(feeder_status)) and (timeout > 0)):
          sleep(time_step)
          timeout = timeout - time_step
    end

    return rq_is_feeder_status_ok(feeder_status)
  end

  def rq_pick_screw(screw_pose, status_input, ready_input, test_in_action=False, approach_dist=10, rotation_speed=rq_pick_rotation_speed,
  pick_speed=25, timeout=rq_feeder_timeout, retract_speed=40, direction=RQ_DIRECTION_CCW, slave_id=9):
      global thread_slave_id = slave_id
      global thread_rotation_speed = rotation_speed
      global thread_direction = direction

      rq_screwdriver_index = rq_comm_slave_id_to_index(slave_id)
      approach_dist_m = norm(approach_dist) / 1000
      pick_speed_m = pick_speed / 1000
      retract_speed_m = retract_speed / 1000
      approach_in_screw_frame = p[0, 0, -approach_dist_m, 0, 0, 0]

      def move_to_approach(screw_pose_in_base_frame, approach_in_screw_frame, blend=True):
        approach_in_base_frame = pose_trans(screw_pose_in_base_frame, approach_in_screw_frame)
        dist_to_approach = point_dist(get_actual_tcp_pose(), approach_in_base_frame)
        offset = 0.005
        blend_radius = offset * 0.99
        if blend and (dist_to_approach > blend_radius):
          approach_to_blend_in_base_frame = pose_trans(approach_in_base_frame, p[0, 0, -offset, 0, 0, 0])
          movel(approach_to_blend_in_base_frame, r=blend_radius)
        else:
          movel(approach_in_base_frame)
        end
      end

      def move_to_retract_servoj(ready_input, robot_speed, slave_id):
        max_distance = 0.05
        linear_speed = -robot_speed
        time_step = 0.008
        initial_pose = get_actual_tcp_pose()
        linear_step = linear_speed * time_step
        distance = 0

        while(get_standard_digital_in(ready_input)):
          distance = distance + linear_step
          next_pose = pose_trans(initial_pose, p[0, 0, distance, 0, 0, 0])
          next_joint_position = get_inverse_kin(next_pose)
          servoj(next_joint_position, t=time_step)

          if (norm(distance) >= max_distance):
            break
          end
        end
        stopj(2)
      end

      def move_to_screw(screw_pose_in_base_frame, robot_speed):
          movel(screw_pose_in_base_frame, v = robot_speed)
      end

      thread start_screwdriver_thread():
        torque_Nm = 1
        rotation_current_mA = floor(torque_Nm * 100)
        rotation_delta_angle = 100
        rotation_timeout_ms = 0
        torque_threshold = 0
        torque_angle_slope = 0
        retries = 40

        rq_set_screw_registers_100x(thread_slave_id, RQ_REGULATION_MODE_SPEED, RQ_ACTIVATE, thread_direction,
        RQ_MODE_NORMAL, RQ_SCREWDRIVER_ON, RQ_TEACHING_OFF, RQ_VACUUM_ON, rotation_current_mA, RQ_MAX_SUPPLY_CURRENT_MA,
        thread_rotation_speed, rotation_delta_angle, rotation_timeout_ms, torque_threshold, torque_angle_slope)

        while (not rq_screwdriver_echo_equal(thread_slave_id, RQ_VACUUM_ON, rotation_current_mA, RQ_SCREWDRIVER_ON,
        thread_direction, thread_rotation_speed, RQ_MODE_NORMAL, RQ_REGULATION_MODE_SPEED, torque_threshold, torque_angle_slope)):
          if ((retries <= 0) or (rq_comm_lost[rq_comm_slave_id_to_index(thread_slave_id)])):
            break
          end
          sleep(0.008)
          rq_set_screw_registers_100x(thread_slave_id, RQ_REGULATION_MODE_SPEED, RQ_ACTIVATE, thread_direction,
          RQ_MODE_NORMAL, RQ_SCREWDRIVER_ON, RQ_TEACHING_OFF, RQ_VACUUM_ON, rotation_current_mA, RQ_MAX_SUPPLY_CURRENT_MA,
           thread_rotation_speed, rotation_delta_angle, rotation_timeout_ms, torque_threshold, torque_angle_slope)
          retries = retries - 1
        end
      end

      def stop_screwdriver(slave_id = 9):
          rotation_current_mA = 0
          rotation_delta_angle = 100
          rotation_timeout_ms = 0
          rotation_speed_rpm = 0
          torque_threshold = 0
          torque_angle_slope = 0

          rq_set_screw_registers_100x(slave_id, RQ_REGULATION_MODE_SPEED, RQ_ACTIVATE, RQ_DIRECTION_CW, RQ_MODE_NORMAL,
          RQ_SCREWDRIVER_OFF, RQ_TEACHING_OFF, RQ_VACUUM_ON, rotation_current_mA, RQ_MAX_SUPPLY_CURRENT_MA,
          rotation_speed_rpm, rotation_delta_angle, rotation_timeout_ms, torque_threshold, torque_angle_slope)

          while (RQ_SCREWDRIVER_ON == rq_get_screw_regulate_echo(slave_id)):
            if(rq_comm_lost[rq_comm_slave_id_to_index(slave_id)]):
              break
            end
            sleep(0.008)
            rq_set_screw_registers_100x(slave_id, RQ_REGULATION_MODE_SPEED, RQ_ACTIVATE, RQ_DIRECTION_CW, RQ_MODE_NORMAL,
            RQ_SCREWDRIVER_OFF,  RQ_TEACHING_OFF, RQ_VACUUM_ON, rotation_current_mA, RQ_MAX_SUPPLY_CURRENT_MA,
            rotation_speed_rpm, rotation_delta_angle, rotation_timeout_ms, torque_threshold, torque_angle_slope)
          end
      end

      def wait_for_screw_present(status_input, ready_input, timeout):
        time_step = 1
        screw_ready = get_standard_digital_in(ready_input)

        while(not screw_ready):
          if (timeout <= 0):
            feeder_status = get_standard_digital_in(status_input)
            if (not feeder_status):
              return RQ_PICK_FAIL_ON_FEEDER_NOT_READY
            end
            return RQ_PICK_FAIL_ON_SCREW_NOT_READY
          end
          sleep(time_step)
          timeout = timeout - time_step
          screw_ready = get_standard_digital_in(ready_input)
        end

        return RQ_FEEDER_SCREW_PRESENT
      end

      thread stop_vacuum_thread():
        rq_set_screw_vacuum(False, thread_slave_id)
         while (RQ_VACUUM_ON == rq_get_screw_vacuum_echo(thread_slave_id)):
           if(rq_comm_lost[rq_comm_slave_id_to_index(thread_slave_id)]):
             break
           end
           sleep(0.008)
           rq_set_screw_vacuum(False, thread_slave_id)
         end
      end

      thread screw_detection():
        global screw_detected_flag = False
        index = rq_comm_slave_id_to_index(thread_slave_id)
        while (not rq_is_screw_detected(thread_slave_id)):
          if(rq_comm_lost[index]):
            break
          end
          global screw_detected_flag = False
          sleep(0.008)
        end
        global screw_detected_flag = not rq_comm_lost[index]
      end

      def start_screw_detection():
        global screw_detected_flag = False
        return run screw_detection()
      end

      def screw_detected():
        return screw_detected_flag
      end

      def wait_for_screw_detected(timeout):
        time_step = 0.1
        detected = False
        thread_id = start_screw_detection()
        while (timeout >= 0):
          sleep(time_step)
          timeout = timeout - time_step
          if (screw_detected()):
            detected = True
            break
          end
        end
        kill thread_id
        return detected
      end

      thread peck():
        while (True):
          movel(pose_trans(get_target_tcp_pose(), p[0, 0, -0.004, 0, 0, 0]), a=0.15, v=0.25)
          movel(pose_trans(get_target_tcp_pose(), p[0, 0, 0.004, 0, 0, 0]), a=0.15, v=0.25)
        end
      end

    #--------------------------------------------------------------------------------------------------
    # Process begins here
    #--------------------------------------------------------------------------------------------------
      if ((not test_in_action) and (rq_wait_for_feeder_status_ok(status_input, timeout))):
        stop_vacuum_thread_id = run stop_vacuum_thread()
        move_to_approach(screw_pose, approach_in_screw_frame)
        join stop_vacuum_thread_id
        if (rq_comm_lost[rq_screwdriver_index]):
          textmsg(RQ_SCREW_FAIL_ON_SCREWDRIVER_COMMUNICATION_LOST_TEXT)

          return RQ_SCREW_FAIL_ON_SCREWDRIVER_COMMUNICATION_LOST
        end
      elif(not rq_is_feeder_status_ok(status_input)):
        sleep(0.008)
        return RQ_PICK_FAIL_ON_FEEDER_NOT_READY
      end

      if ((not rq_is_feeder_screw_ready(ready_input)) and (rq_wait_for_feeder_status_ok(status_input, timeout))):
        move_to_approach(screw_pose, approach_in_screw_frame, blend=False)
      elif(not rq_is_feeder_status_ok(status_input)):
        return RQ_PICK_FAIL_ON_FEEDER_NOT_READY
      end

      feeder_result = wait_for_screw_present(status_input, ready_input, timeout)
      if (RQ_FEEDER_SCREW_PRESENT != feeder_result):
          return feeder_result
      end

      start_screwdriver_thread_id = run start_screwdriver_thread()
      move_to_screw(screw_pose, pick_speed_m)
      join start_screwdriver_thread_id

      if (rq_comm_lost[rq_screwdriver_index]):
        textmsg(RQ_SCREW_FAIL_ON_SCREWDRIVER_COMMUNICATION_LOST_TEXT)
        kill start_screwdriver_thread_id

        return RQ_SCREW_FAIL_ON_SCREWDRIVER_COMMUNICATION_LOST
      end

      if (not rq_screwdriver_is_activated(slave_id)):
        return RQ_PICK_FAIL_ON_SCREWDRIVER_NOT_ACTIVATED
      end

      peck_thread_id = run peck()
      wait_for_screw_detected(2)
      kill peck_thread_id
      move_to_retract_servoj(ready_input, retract_speed_m, slave_id)
      is_screw_detected = wait_for_screw_detected(2)
      stop_screwdriver(slave_id)

      if (rq_comm_lost[rq_screwdriver_index]):
        textmsg(RQ_SCREW_FAIL_ON_SCREWDRIVER_COMMUNICATION_LOST_TEXT)

        return RQ_SCREW_FAIL_ON_SCREWDRIVER_COMMUNICATION_LOST
      end
      if (not is_screw_detected):
          return RQ_PICK_FAIL_ON_SCREW_NOT_DETECTED
      end

      return RQ_PICK_SUCCESS
  end
  global rq_screwdriver_faults = [0,0,0,0,0,0,0,0]
  global rq_max_thread_contact_distance = 0.05
  global rq_unhandled_error = RQ_NO_FAULT
  global rq_fs_speed = 0.008
  global rq_log_screwing = False
  copilot_kinematics_rpc_server = rpc_factory("xmlrpc","http://localhost:4251/")
  global app_time = 0
  global rq_find_surface_time = 0
  global rq_screwing_time = 0

  thread app_timer():
    step_time = get_steptime()
    app_time = 0
    while(True):
      app_time = app_time + step_time
      sleep(step_time)
    end
  end

  def rq_screw(operation_mode, regulation_mode, rotation_current, rotation_speed, rotation_angle, timeout, teaching,
  torque_threshold, torque_angle_slope, direction=RQ_DIRECTION_CW, slave_id=9):
    direction = direction
    activation = RQ_ACTIVATE
    regulate = RQ_SCREWDRIVER_ON
    vacuum = rq_get_screw_vacuum_echo(slave_id)
    rotation_speed_raw = rotation_speed
    max_supply_current = RQ_MAX_SUPPLY_CURRENT_MA
    time_max = timeout * 1000
    index = rq_comm_slave_id_to_index(slave_id)

    if(timeout == RQ_UNUSED_PARAMETER):
      time_max = RQ_ENDLESS_TIMEOUT
    end

    retries = 40
    rq_set_screw_registers_100x(slave_id, regulation_mode, activation, direction, operation_mode, regulate, teaching, vacuum,
                                rotation_current, max_supply_current, rotation_speed_raw, rotation_angle, time_max,
                                torque_threshold, torque_angle_slope)
    while (not rq_screwdriver_echo_equal(slave_id, vacuum, rotation_current, regulate, direction, rotation_speed_raw, operation_mode, regulation_mode, torque_threshold, torque_angle_slope)):
      if ((retries <= 0) or (rq_comm_lost[index])):
        return False
      end
      sleep(0.008)
      rq_set_screw_registers_100x(slave_id, regulation_mode, activation, direction, operation_mode, regulate, teaching, vacuum,
                                  rotation_current, max_supply_current, rotation_speed_raw, rotation_angle, time_max,
                                  torque_threshold, torque_angle_slope)
      retries = retries - 1
    end
     return True
  end

  def rq_screw_with_force(operation_mode, regulation_mode, rotation_current, rotation_speed, rotation_angle,
  teach_thread_mating_position, teach_final_position, teaching, torque_threshold, torque_angle_slope, force=10,
  timeout=10, distance_tolerance=0, direction=RQ_DIRECTION_CW, slave_id=9):
    app_timer_id = -1
    if(rq_log_screwing):
      app_timer_id = run app_timer()
    end

    def kill_app_timer(app_timer_id):
      if(rq_log_screwing):
        kill app_timer_id
      end
    end

    thread action_status_thread():
      while (True):
        thread_action_status = rq_get_screw_action(thread_slave_id)
        if (rq_comm_lost[rq_comm_slave_id_to_index(thread_slave_id)]):
          break
        end
      end
    end

    global find_surface_turn_direction = direction
    thread start_find_surface_screwdriver():
      rq_screw_turn(regulation_mode=RQ_REGULATION_MODE_SPEED, torque_Nm=1, rotation_angle=0, rotation_speed_rpm=100, direction=not find_surface_turn_direction, slave_id=thread_slave_id)
    end

    def is_enabled(parameter):
      return parameter > RQ_UNUSED_PARAMETER
    end

    global thread_slave_id = slave_id
    rq_unhandled_error = RQ_NO_FAULT
    rq_screwdriver_index = rq_comm_slave_id_to_index(slave_id)

    global rq_actual_thread_mating_position = get_actual_tcp_pose()

    if (rq_is_comm_lost(slave_id)):
      textmsg(RQ_SCREW_FAIL_ON_SCREWDRIVER_COMMUNICATION_LOST_TEXT)
      rq_unhandled_error = RQ_SCREW_FAIL_ON_SCREWDRIVER_COMMUNICATION_LOST
      kill_app_timer(app_timer_id)

      return RQ_SCREW_FAIL_ON_SCREWDRIVER_COMMUNICATION_LOST
    end

    activation_and_screw_detection_registers = rq_get_activation_and_screw_detection(slave_id)

    if (not activation_and_screw_detection_registers[0]):
      textmsg(RQ_NOT_ACTIVATED_MESSAGE)
      kill_app_timer(app_timer_id)

      return RQ_SCREW_FAIL_ON_SCREWDRIVER_NOT_ACTIVATED
    end

    if(not activation_and_screw_detection_registers[1]):
      textmsg(RQ_SCREW_FAIL_ON_NO_SCREW_TEXT)
      kill_app_timer(app_timer_id)

      return RQ_SCREW_FAIL_ON_SCREW_NOT_DETECTED
    end

    before_find_surface_time = app_time
    start_find_surface_screwdriver_id = run start_find_surface_screwdriver()

    success = rq_wait_for_contact_with_thread(rq_max_thread_contact_distance, rq_fs_speed)
    if (not success):
      kill start_find_surface_screwdriver_id
      rq_screw_stop()
      textmsg(RQ_SCREW_FAIL_ON_CONTACT_NOT_FOUND_TEXT)
      rq_unhandled_error = RQ_SCREW_FAIL_ON_CONTACT_NOT_FOUND
      kill_app_timer(app_timer_id)

      return RQ_SCREW_FAIL_ON_CONTACT_NOT_FOUND
    end

    rq_find_surface_time = app_time - before_find_surface_time

    kill start_find_surface_screwdriver_id

    rq_actual_thread_mating_position = get_actual_tcp_pose()

    if(not rq_is_screw_detected(slave_id)):
      rq_screw_stop()
      textmsg(RQ_SCREW_FAIL_ON_NO_SCREW_TEXT)
      kill_app_timer(app_timer_id)

      return RQ_SCREW_FAIL_ON_SCREW_NOT_DETECTED
    end

    before_screwing_time = app_time
    result = rq_screw(operation_mode, regulation_mode, rotation_current, rotation_speed, rotation_angle, timeout,
    teaching, torque_threshold, torque_angle_slope, direction, slave_id)
    if (result == False):
      if (rq_comm_lost[rq_screwdriver_index]):
        textmsg(RQ_SCREW_FAIL_ON_SCREWDRIVER_COMMUNICATION_LOST_TEXT)
        rq_unhandled_error = RQ_SCREW_FAIL_ON_SCREWDRIVER_COMMUNICATION_LOST
        kill_app_timer(app_timer_id)

        return RQ_SCREW_FAIL_ON_SCREWDRIVER_COMMUNICATION_LOST
      else:
        textmsg(RQ_SCREW_FAIL_ON_SCREWDRIVER_NOT_RESPONDING_TEXT)
        rq_unhandled_error = RQ_SCREW_FAIL_ON_SCREWDRIVER_NOT_RESPONDING
        rq_screw_stop()
        kill_app_timer(app_timer_id)

        return RQ_SCREW_FAIL_ON_SCREWDRIVER_NOT_RESPONDING
      end

    end
    global thread_action_status = RQ_IN_ACTION
    action_status_thread_id = run action_status_thread()

    rq_speed_slider = copilot_kinematics_rpc_server.gettargetspeedfraction()
    if(rq_speed_slider < 1.0):
      copilot_kinematics_rpc_server.settargetspeedfraction(1.0)
    end

    follow_time_step = 0.008

    force_node_thread_id = rq_setup_screw_force(force)

    teach_final_pose_in_thread_frame = pose_trans(pose_inv(teach_thread_mating_position), teach_final_position)

    while (thread_action_status == RQ_IN_ACTION):
      sleep(follow_time_step)
      if (rq_comm_lost[rq_screwdriver_index]):
        kill action_status_thread_id
        kill force_node_thread_id
        kill_app_timer(app_timer_id)

        textmsg(RQ_SCREW_FAIL_ON_SCREWDRIVER_COMMUNICATION_LOST_TEXT)
        rq_unhandled_error = RQ_SCREW_FAIL_ON_SCREWDRIVER_COMMUNICATION_LOST
        copilot_kinematics_rpc_server.settargetspeedfraction(rq_speed_slider)

        return RQ_SCREW_FAIL_ON_SCREWDRIVER_COMMUNICATION_LOST
      end

      if(is_enabled(distance_tolerance)):
        tool_position = get_actual_tcp_pose()
        actual_tool_pose_in_thread_frame = pose_trans(pose_inv(rq_actual_thread_mating_position), tool_position)

        position_delta = actual_tool_pose_in_thread_frame[2] - teach_final_pose_in_thread_frame[2]

        if(position_delta > (distance_tolerance / RQ_MILLI_UNIT_TO_UNIT_FACTOR)):
          copilot_kinematics_rpc_server.settargetspeedfraction(rq_speed_slider)

          kill action_status_thread_id
          kill force_node_thread_id
          kill_app_timer(app_timer_id)

          rq_screw_stop()
          textmsg(RQ_SCREW_FAIL_ON_DISTANCE_MAX_TEXT)

          return RQ_SCREW_FAIL_ON_DISTANCE_MAX
        end
      end
    end

    rq_screwing_time = app_time - before_screwing_time
    if(rq_speed_slider < 1.0):
      copilot_kinematics_rpc_server.settargetspeedfraction(rq_speed_slider)
    end

    kill action_status_thread_id
    kill force_node_thread_id

    if (rq_comm_lost[rq_screwdriver_index]):
      textmsg(RQ_SCREW_FAIL_ON_SCREWDRIVER_COMMUNICATION_LOST_TEXT)
      rq_unhandled_error = RQ_SCREW_FAIL_ON_SCREWDRIVER_COMMUNICATION_LOST
      kill_app_timer(app_timer_id)

      return RQ_SCREW_FAIL_ON_SCREWDRIVER_COMMUNICATION_LOST
    end

    rq_screwdriver_faults = rq_get_screw_fault()
    rq_log_application_warning(rq_screwdriver_faults)
    actual_final_position = get_actual_tcp_pose()

    kill_app_timer(app_timer_id)

    return rq_get_screw_with_force_result(regulation_mode, thread_action_status,
    teach_thread_mating_position, teach_final_position, rq_actual_thread_mating_position, actual_final_position,
    distance_tolerance, timeout, rq_screwdriver_faults)
  end

  #--------------------------------------------------------------------------------------------------
  # Returns screw with a clutch result
  #
  #    action_status          : action status from screwdriver
  #    time                   : elapsed time
  #    time_max               : maximum time elapsed to deem screw operation successful
  #    distance_tolerance     : distance tolerance wanted
  #    rotations_tolerance    : number of rotations wanted
  #    rotations_min          : minimum number of rotations to deem screw operation successful
  #    rotations_max          : maximum number of rotations to deem screw operation successful
  #
  #--------------------------------------------------------------------------------------------------
  def rq_get_screw_with_force_result(regulation_mode, action_status, teach_thread_mating_position,
  teach_final_position, actual_thread_mating_position, actual_final_position, distance_tolerance, timeout, screwdriver_faults):

    def is_enabled(parameter):
        return parameter > RQ_UNUSED_PARAMETER
    end

    teach_final_pose_in_thread_frame = pose_trans(pose_inv(teach_thread_mating_position), teach_final_position)
    actual_final_pose_in_thread_frame = pose_trans(pose_inv(actual_thread_mating_position), actual_final_position)

    position_delta = actual_final_pose_in_thread_frame[2] - teach_final_pose_in_thread_frame[2]

    if(is_enabled(timeout) and timeout > 0 and rq_is_timeout_cause()):
      return RQ_SCREW_FAIL_ON_TIME_MAX
    elif(is_enabled(distance_tolerance) and (position_delta > (distance_tolerance / RQ_MILLI_UNIT_TO_UNIT_FACTOR))):
      return RQ_SCREW_FAIL_ON_DISTANCE_MAX
    elif(is_enabled(distance_tolerance) and (position_delta < -(distance_tolerance / RQ_MILLI_UNIT_TO_UNIT_FACTOR))):
      return RQ_SCREW_FAIL_ON_DISTANCE_MIN
    elif(rq_screwdriver_in_fault(screwdriver_faults)):
      textmsg("Faults : ", screwdriver_faults)
      return RQ_SCREW_FAIL_ON_UNHANDLED_ERROR
    elif(action_status == RQ_NO_DETECTION):
      textmsg(RQ_SCREW_FAIL_WITHOUT_DETECTION_TEXT)
      rq_unhandled_error = RQ_SCREW_FAIL_WITHOUT_DETECTION
      return RQ_SCREW_FAIL_WITHOUT_DETECTION
    else:
      return RQ_SCREW_SUCCESS
    end
  end

  def rq_log_application_warning(screwdriver_faults):

     if(not rq_screwdriver_in_fault(screwdriver_faults)):
      rq_application_warning_message = RQ_NO_FAULT_MESSAGE
      textmsg(RQ_NO_FAULT_MESSAGE)
     end

     if(screwdriver_faults[0] > 0):
       rq_warning_prefix = "Application warnings : "
       rq_fault_separator = ", "
       rq_application_warning = integer_to_binary_list(screwdriver_faults[0])

       if(rq_application_warning[0]):
         rq_application_warning_message = str_cat(rq_warning_prefix, RQ_COMMUNICATION_NOT_READY_MESSAGE)
         textmsg(rq_application_warning_message)
       end
       if(rq_application_warning[1]):
         rq_application_warning_message = str_cat(rq_warning_prefix, RQ_BLOCKED_AT_START_MESSAGE)
         textmsg(rq_application_warning_message)
       end
       if(rq_application_warning[2]):
         rq_application_warning_message = str_cat(rq_warning_prefix, RQ_RESTRICTION_BEFORE_ANGLE_MESSAGE)
         textmsg(rq_application_warning_message)
       end
       if(rq_application_warning[3]):
         rq_application_warning_message = str_cat(rq_warning_prefix, RQ_TIMEOUT_MESSAGE)
         textmsg(rq_application_warning_message)
       end
       if(rq_application_warning[4]):
         rq_application_warning_message = str_cat(rq_warning_prefix, RQ_REGULATION_WHILE_NOT_ACT_MESSAGE)
         textmsg(rq_application_warning_message)
       end
       if(rq_application_warning[5]):
        rq_application_warning_message = str_cat(rq_warning_prefix, RQ_NOT_ACTIVATED_MESSAGE)
        textmsg(rq_application_warning_message)
       end
        if(rq_application_warning[6]):
         rq_application_warning_message = str_cat(rq_warning_prefix, "Over torque")
         textmsg(rq_application_warning_message)
        end
        if(rq_application_warning[7]):
         rq_application_warning_message = str_cat(rq_warning_prefix, "Under torque")
         textmsg(rq_application_warning_message)
        end
        if(rq_application_warning[8]):
         rq_application_warning_message = str_cat(rq_warning_prefix, "Processing recorded data failed")
         textmsg(rq_application_warning_message)
        end
        if(rq_application_warning[9]):
         rq_application_warning_message = str_cat(rq_warning_prefix, "Torque parameters out of bounds")
         textmsg(rq_application_warning_message)
        end
     end
  end

  def rq_screwdriver_in_fault(screwdriver_faults):
    index = 0
    while (index < get_list_length(screwdriver_faults)):
     if(screwdriver_faults[index] > 0):
       return True
     end
     index = index + 1
    end

    return False
  end

  def rq_get_screwdriver_faults_message():
    if(rq_screwdriver_faults[0] == 0):
      return str_cat("Screwdriver faults code : ", to_str(rq_screwdriver_faults))
    end
    rq_application_warning_message = "Application warnings : "
    rq_fault_separator = "<br>"
    rq_application_warning = integer_to_binary_list(rq_screwdriver_faults[0])

    if(rq_application_warning[0]):
         rq_application_warning_message = str_cat(rq_application_warning_message, RQ_COMMUNICATION_NOT_READY_MESSAGE)
    end
    if(rq_application_warning[1]):
      rq_application_warning_message = str_cat(rq_application_warning_message, rq_fault_separator)
      rq_application_warning_message = str_cat(rq_application_warning_message, RQ_BLOCKED_AT_START_MESSAGE)
    end
    if(rq_application_warning[2]):
      rq_application_warning_message = str_cat(rq_application_warning_message, rq_fault_separator)
      rq_application_warning_message = str_cat(rq_application_warning_message, RQ_RESTRICTION_BEFORE_ANGLE_MESSAGE)
    end
    if(rq_application_warning[3]):
      rq_application_warning_message = str_cat(rq_application_warning_message, rq_fault_separator)
      rq_application_warning_message = str_cat(rq_application_warning_message, RQ_TIMEOUT_MESSAGE)
    end
    if(rq_application_warning[4]):
      rq_application_warning_message = str_cat(rq_application_warning_message, rq_fault_separator)
      rq_application_warning_message = str_cat(rq_application_warning_message, RQ_REGULATION_WHILE_NOT_ACT_MESSAGE)
    end
    if(rq_application_warning[5]):
      rq_application_warning_message = str_cat(rq_application_warning_message, rq_fault_separator)
      rq_application_warning_message = str_cat(rq_application_warning_message, RQ_NOT_ACTIVATED_MESSAGE)
    end
    return rq_application_warning_message
  end

  def rq_is_blocked_at_start_cause():
    rq_application_warning = integer_to_binary_list(rq_screwdriver_faults[0])

    return rq_application_warning[1]
  end

  def rq_is_restricted_before_angle_cause():
    rq_application_warning = integer_to_binary_list(rq_screwdriver_faults[0])

    return rq_application_warning[2]
  end

  def rq_is_timeout_cause():
    rq_application_warning = integer_to_binary_list(rq_screwdriver_faults[0])

    return rq_application_warning[3]
  end

  def rq_is_communication_lost_cause():
    return rq_unhandled_error == RQ_SCREW_FAIL_ON_SCREWDRIVER_COMMUNICATION_LOST
  end

  def rq_is_screwdriver_wrong_echo_cause():
    return rq_unhandled_error == RQ_SCREW_FAIL_ON_SCREWDRIVER_NOT_RESPONDING
  end

  def rq_is_contact_not_found_cause():
    return rq_unhandled_error == RQ_SCREW_FAIL_ON_CONTACT_NOT_FOUND
  end

  def rq_is_action_finished_without_detection_cause():
    return rq_unhandled_error == RQ_SCREW_FAIL_WITHOUT_DETECTION
  end

  #--------------------------------------------------------------------------------------------------
  # Turns the screwdriver at the specified speed and torque
  #
  #    regulation_mode        : Regulation mode (default RQ_REGULATION_MODE_SPEED)
  #    torque_Nm              : Torque value in Nm (default 1 Nm)
  #    rotation_angle         : Rotation angle in deg (default 0 deg)
  #    rotation_speed_rpm     : Rotation speed in rpm (default 100 rpm)
  #    direction              : Rotation direction (RQ_DIRECTION_CCW = True, RQ_DIRECTION_CW = False) (default RQ_DIRECTION_CW)
  #    slave_id               : slave id of the screwdriver (default 9)
  #
  #--------------------------------------------------------------------------------------------------
  def rq_screw_turn(regulation_mode=RQ_REGULATION_MODE_SPEED, torque_Nm=1, rotation_angle=0, rotation_speed_rpm=100, direction=RQ_DIRECTION_CW, slave_id=9):
      activation = RQ_ACTIVATE
      operation_mode = RQ_MODE_NORMAL
      regulate = RQ_SCREWDRIVER_ON
      vacuum = rq_get_screw_vacuum_echo(slave_id)
      rotation_current = floor(torque_Nm * 100)
      rotation_speed_raw = floor(rotation_speed_rpm)
      max_supply_current = RQ_MAX_SUPPLY_CURRENT_MA
      time_max = 0
      torque_threshold = 0
      torque_angle_slope = 0

      rq_set_screw_registers_100x(slave_id, regulation_mode, activation, direction, operation_mode, regulate, RQ_TEACHING_OFF, vacuum,
      rotation_current, max_supply_current, rotation_speed_raw, rotation_angle, time_max, torque_threshold, torque_angle_slope)
  end

  #--------------------------------------------------------------------------------------------------
  # Stops the screwdriver
  #
  #    slave_id               : slave id of the screwdriver (default 9)
  #
  #--------------------------------------------------------------------------------------------------
  def rq_screw_stop(slave_id = 9):
      rq_set_screw_regulate(slave_id, False)
  end

  def rq_stop_regulating_and_stop_vacuum(slave_id = 9):
      thread_slave_id = slave_id
      thread stop_vacuum():
        rq_screw_vacuum_off_and_stop_regulate(thread_slave_id)
      end
      run stop_vacuum()
  end
  def rq_update_window_with_next_value(new_value, window):
     i = 0
     while(i < length(window) - 1):
       window[i] = window[i + 1]
       i = i + 1
     end
     window[length(window) - 1] = new_value
     return window
  end
  def rq_average(window):
     sum = 0
     i = 0
     while(i < length(window)):
       sum = sum + window[i]
       i = i + 1
     end
     return sum/length(window)
  end
  def rq_are_all_values_positive(window):
    i = 0
    while(i < length(window)):
      if (window[i] <= 0):
        return 0
      end
      i = i + 1
    end
    return 1
  end

  global rq_z_window = [0, 0, 0, 0, 0, 0, 0, 0, 0, 0]
  global rq_dz_window = [0, 0, 0, 0, 0, 0, 0, 0, 0, 0]
  global rq_z_avg_last = 0
  def rq_compute_next_z_avg(new_z):
    rq_z_window = rq_update_window_with_next_value(new_z, rq_z_window)
    return rq_average(rq_z_window)
  end
  def rq_compute_stop_signal(new_dz):
    rq_dz_window = rq_update_window_with_next_value(new_dz, rq_dz_window)
    return rq_are_all_values_positive(rq_dz_window)
  end

  thread rq_auto_stop():
    counter = 0
    stop_signal = 0
    starting_frame = pose_inv(get_actual_tcp_pose())
    while(get_flag(0)):
      pose = pose_trans(starting_frame, get_actual_tcp_pose())
      z = pose[2]
      z_avg = rq_compute_next_z_avg(z)
      dz = z_avg - rq_z_avg_last
      if (counter > length(rq_z_window)):
        stop_signal = rq_compute_stop_signal(dz)
        if (stop_signal):
          set_flag(0, False)
        end
      end
      rq_z_avg_last = z_avg
      counter = counter + 1
      sleep(0.008)
    end
  end

  def rq_unscrew(direction, force=5, rotation_speed_rpm=100, torque_Nm=4, unscrew_stiffness = [100, 100, 70, 100, 100, 100], unscrew_adaptive_stiffness = True, slave_id=9):
    result = rq_screw_start_force_control_tool_z(force)
    thread_id = result[0]
    force_node_id = result[1]
    rotation_current_mA = floor(torque_Nm * 100)

    node_rpc_server.setforcecontrolstiffness(force_node_id, unscrew_stiffness)
    node_rpc_server.setforcecontroladaptivestiffnessenabledaxes(force_node_id, unscrew_adaptive_stiffness)

    vacuum = rq_get_screw_vacuum_echo(slave_id)

    rq_set_screw_registers_100x(slave_id, RQ_REGULATION_MODE_SPEED, RQ_ACTIVATE, direction, RQ_MODE_NORMAL,
    RQ_SCREWDRIVER_ON, RQ_TEACHING_OFF, vacuum, rotation_current_mA, RQ_MAX_SUPPLY_CURRENT_MA, rotation_speed_rpm,
    0, 0, 0, 0)

    return thread_id
  end

  def rq_wait_for_interruption(slave_id = 9):
    while(get_flag(0) and (rq_get_screw_action(slave_id) == RQ_IN_ACTION)):
      sleep(0.008)
    end
  end

  def rq_unscrew_stop(thread_id, tcp_pose_before_unscrew, slave_id=9):
    vacuum = rq_get_screw_vacuum_echo(slave_id)
    rq_set_screw_registers_100x(slave_id, RQ_REGULATION_MODE_SPEED, RQ_ACTIVATE, RQ_DIRECTION_CW, RQ_MODE_NORMAL,
    RQ_SCREWDRIVER_OFF, RQ_TEACHING_OFF, vacuum, 0, RQ_MAX_SUPPLY_CURRENT_MA, 0, 0, 0, 0, 0)
    rq_screw_stop_force_control(thread_id)
    turns_to_unscrew = rq_get_screw_delta_angle_deg(slave_id)/360
    tcp_pose_after_unscrew = get_actual_tcp_pose()
    distance_to_unscrew = point_dist(tcp_pose_before_unscrew, tcp_pose_after_unscrew) * 1000
    pitch_estimated = distance_to_unscrew/turns_to_unscrew
  end

  def rq_wait_nb_turns(nb_turns=2, slave_id=9):
    time_step_ms = 0.1
    timeout_ms = 2000
    remaining_retries = timeout_ms / time_step_ms
    minimum_nb_degrees = rq_get_screw_delta_angle_deg(slave_id) + nb_turns * 360

    while(rq_get_screw_delta_angle_deg(slave_id) < minimum_nb_degrees and remaining_retries > 0):
      sleep(time_step_ms)
      remaining_retries = remaining_retries - 1
    end
  end

  def rq_auto_unscrew(direction=RQ_DIRECTION_CCW, rotation_speed=100):
    tcp_pose_before_unscrew = get_actual_tcp_pose()
    thread_id = rq_unscrew(direction,rotation_speed_rpm=rotation_speed)
    rq_wait_nb_turns()
    set_flag(0, True)
    auto_stop_thread_id = run rq_auto_stop()
    rq_wait_for_interruption()
    rq_unscrew_stop(thread_id, tcp_pose_before_unscrew)
    join auto_stop_thread_id
  end
  def rq_screw_start_force_control_tool_z(target_force_z = 10):
      return rq_screw_start_force_control(force_control_enabled_axes = [False, False, True, False, False, False], target_force = [0, 0, target_force_z, 0, 0, 0], max_negative_deviation = [0, 0, -0.1, 0, 0, 0], max_positive_deviation = [0, 0, 0.1, 0, 0, 0])
  end
  def rq_screw_start_force_control_tool_z_with_xy_compliance(target_force_z = 10):
      return rq_screw_start_force_control(force_control_enabled_axes = [True, True, True, False, False, False], target_force = [0, 0, target_force_z, 0, 0, 0], max_negative_deviation = [-1, -1, -1, 0, 0, 0], max_positive_deviation = [1, 1, 1, 0, 0, 0])
  end
  def rq_screw_start_scara_mode():
      return rq_screw_start_scara_with_force(target_force_z = 0)
  end
  def rq_screw_start_scara_with_force(target_force_z = 10):
      return rq_screw_start_force_control(force_control_enabled_axes = [True, True, True, False, False, False], target_force = [0, 0, target_force_z, 0, 0, 0], max_negative_deviation = [-0.5, -0.5, -0.5, 0, 0, 0], max_positive_deviation = [0.5, 0.5, 0.5, 0, 0, 0])
  end
  def rq_screw_start_force_control(force_control_enabled_axes = [False, False, False, False, False, False], target_force = [0, 0, 0, 0, 0, 0], max_negative_deviation = [0, 0, 0, 0, 0, 0], max_positive_deviation = [0, 0, 0, 0, 0, 0], stiffness = [100, 100, 100, 100, 100, 100], adaptive_stiffness = True):
      RELATIVE_TO_TCP = 1
      force_node_id = node_rpc_server.createnewforcenode()
      servoj_node_id = node_rpc_server.createnewservojnode()
      node_rpc_server.setparentid(servoj_node_id, force_node_id)
      node_rpc_server.setforcecontrolfeature(force_node_id, RELATIVE_TO_TCP)
      node_rpc_server.setforcecontrolenabledaxes(force_node_id, force_control_enabled_axes)
      node_rpc_server.setforcecontroltargetforce(force_node_id, target_force)
      node_rpc_server.setforcecontrolmaximaldeviation(force_node_id, max_negative_deviation, max_positive_deviation)
      node_rpc_server.setforcecontrolstiffness(force_node_id, stiffness)
      node_rpc_server.setforcecontroladaptivestiffnessenabledaxes(force_node_id, adaptive_stiffness)
      # This moveJ is used to prevent "another thread is already controlling the robot error"
      movej(get_actual_joint_positions())
      set_servoj_node_cmd(get_actual_joint_positions())
      reset_node_executor()
      active_and_reset_node(force_node_id)
      active_and_reset_node(servoj_node_id)
      zero_ftsensor()

      return [run execute_node_thread(), force_node_id]
  end
  def rq_screw_stop_force_control(node_execution_thread):
      kill_thread(node_execution_thread)
  end
  def rq_setup_screw_force(force):
    def concat(str1, str2, str3):
      return str_cat(str1, str_cat(str2, str3))
    end
    def key_val(key, val):
      return concat(concat("`", key, "`"), ":", val)
    end
    def json_force_node(force):
      json = "{"
      json = concat(json, key_val("forceFrame", 1), ",")
      json = concat(json, key_val("isAdaptive", "true"), ",")
      json = concat(json, key_val("isForceControlAboutActualPosition", "true"), ",")
      json = concat(json, key_val("isForceMode", "[false,false,true,false,false,false]"), ",")
      json = concat(json, key_val("maxNegativeDeviation", [0,0,-0.01,0,0,0]), ",")
      json = concat(json, key_val("maxPositiveDeviation", [0,0,0.1,0,0,0]), ",")
      json = concat(json, key_val("stiffness", [0,0,0.8,0,0,0]), ",")
      json = concat(json, key_val("targetTcpWrench", [0,0,force,0,0,0]), "}")
      return json
    end
    def init_force_node(force):
      movej(get_actual_joint_positions()) # This moveJ is used to prevent "another thread is already controlling the robot error".
      force_node_id = node_rpc_server.createnewforcenode()
      node_rpc_server.fromjson(force_node_id, json_force_node(force))
      reset_node_executor()
      active_and_reset_node(force_node_id)
      node_execution_thread = run execute_node_thread()
      return node_execution_thread
    end
    # initialize forcenode: adapt to direction
    node_execution_thread = init_force_node(force)
    return node_execution_thread
  end
  def rq_wait_for_contact_with_thread(max_distance, wanted_speed = 0.004):
    zero_ftsensor()

    return rq_linear_search_urcap(direction="Z+", force_threshold = 10, speed = wanted_speed, max_distance = max_distance, feature = 1)
  end
  def rq_extract_value_from_register_value(register_value, first_bit, total_of_bit):
      register_binary_list = integer_to_binary_list(register_value)
      bit_exponent = 0
      value = 0
      next_bit = first_bit
      last_bit = first_bit + total_of_bit

      while(next_bit < last_bit):
          if(register_binary_list[next_bit]):
              value = value + pow(2,bit_exponent)
          end
          next_bit = next_bit + 1
          bit_exponent = bit_exponent + 1
      end

      return value
  end

  def rq_extract_boolean_from_register_value(register_value, bit_number):
      register_binary_list = integer_to_binary_list(register_value)
      return register_binary_list[bit_number]
  end

  def rq_insert_boolean_in_register_value(register_value, bit_number, boolean_value):
      register_binary_list = integer_to_binary_list(register_value)
      register_binary_list[bit_number] = boolean_value
      return binary_list_to_integer(register_binary_list)
  end

  def rq_insert_lsb_in_register_value(register_value, byte_value):
      return rq_insert_value_in_register_value(register_value, 0, 8, byte_value)
  end

  def rq_insert_msb_in_register_value(register_value, byte_value):
      return rq_insert_value_in_register_value(register_value, 8, 8, byte_value)
  end

  def rq_insert_value_in_register_value(register_value, first_bit, total_of_bit, value):
      register_binary_list = integer_to_binary_list(register_value)
      value_list = integer_to_binary_list(value)
      next_value_bit = 0
      next_register_value_bit = first_bit
      last_bit = first_bit + total_of_bit

      while(next_register_value_bit < last_bit):
          register_binary_list[next_register_value_bit] = value_list[next_value_bit]
          next_register_value_bit = next_register_value_bit + 1
          next_value_bit = next_value_bit + 1
      end

      return binary_list_to_integer(register_binary_list)
  end
  RQ_READ_SCREWDRIVER_REGISTERS_SIZE = 22

  rq_xml_rpc_modbus = rpc_factory("xmlrpc", "http://127.0.0.1:8090/")
  rq_xml_rpc_modbus_debug = rpc_factory("xmlrpc", "http://127.0.0.1:8090/")

  rq_comm_slave_ids = [9]

  global rq_comm_lost = [False, False, False, False]

  rq_comm_write_3_registers_100x_request = [False, False, False, False]
  rq_comm_write_8_registers_100x_request = [False, False, False, False]
  rq_comm_write_register_1000 = [0, 0, 0, 0]
  rq_comm_write_register_1001 = [0, 0, 0, 0]
  rq_comm_write_register_1002 = [0, 0, 0, 0]
  rq_comm_write_register_1003 = [0, 0, 0, 0]
  rq_comm_write_register_1004 = [0, 0, 0, 0]
  rq_comm_write_register_1005 = [0, 0, 0, 0]
  rq_comm_write_register_1006 = [0, 0, 0, 0]
  rq_comm_write_register_1007 = [0, 0, 0, 0]

  rq_comm_write_register_6020_request = [False, False, False, False]
  rq_comm_write_register_6020 = [0, 0, 0, 0]

  rq_comm_read_3_registers_200x_request = [False, False, False, False]
  rq_comm_read_22_registers_200x_request = [False, False, False, False]
  rq_comm_read_register_2000 = [0, 0, 0, 0]
  rq_comm_read_register_2001 = [0, 0, 0, 0]
  rq_comm_read_register_2002 = [0, 0, 0, 0]
  rq_comm_read_register_2003 = [0, 0, 0, 0]
  rq_comm_read_register_2004 = [0, 0, 0, 0]
  rq_comm_read_register_2005 = [0, 0, 0, 0]
  rq_comm_read_register_2006 = [0, 0, 0, 0]
  rq_comm_read_register_2007 = [0, 0, 0, 0]
  rq_comm_read_register_2008 = [0, 0, 0, 0]
  rq_comm_read_register_2009 = [0, 0, 0, 0]
  rq_comm_read_register_2010 = [0, 0, 0, 0]
  rq_comm_read_register_2011 = [0, 0, 0, 0]
  rq_comm_read_register_2012 = [0, 0, 0, 0]
  rq_comm_read_register_2013 = [0, 0, 0, 0]
  rq_comm_read_register_2014 = [0, 0, 0, 0]
  rq_comm_read_register_2015 = [0, 0, 0, 0]
  rq_comm_read_register_2016 = [0, 0, 0, 0]
  rq_comm_read_register_2017 = [0, 0, 0, 0]
  rq_comm_read_register_2018 = [0, 0, 0, 0]
  rq_comm_read_register_2019 = [0, 0, 0, 0]
  rq_comm_read_register_2020 = [0, 0, 0, 0]
  rq_comm_read_register_2021 = [0, 0, 0, 0]

  rq_comm_read_registers_250x_request = [False, False, False, False]
  rq_comm_read_register_2500 = [0, 0, 0, 0]
  rq_comm_read_register_2501 = [0, 0, 0, 0]
  rq_comm_read_register_2502 = [0, 0, 0, 0]
  rq_comm_read_register_2503 = [0, 0, 0, 0]
  rq_comm_read_register_2504 = [0, 0, 0, 0]
  rq_comm_read_register_2505 = [0, 0, 0, 0]
  rq_comm_read_register_2506 = [0, 0, 0, 0]
  rq_comm_read_register_2507 = [0, 0, 0, 0]
  rq_comm_read_register_2508 = [0, 0, 0, 0]

  rq_comm_read_3_registers_602x_request = [False, False, False, False]
  rq_comm_read_register_6020 = [0, 0, 0, 0]
  rq_comm_read_register_6021 = [0, 0, 0, 0]
  rq_comm_read_register_6022 = [0, 0, 0, 0]

  def rq_comm_write_registers_100x(slave_id, registers_100x, number_of_registers):
      if(number_of_registers == 3):
          enter_critical
              index = rq_comm_slave_id_to_index(slave_id)
              rq_comm_write_register_1000[index] = registers_100x[0]
              rq_comm_write_register_1001[index] = registers_100x[1]
              rq_comm_write_register_1002[index] = registers_100x[2]
              rq_comm_write_3_registers_100x_request[index] = True
          exit_critical

          while(rq_comm_write_3_registers_100x_request[index]):
              sleep(0.008)
          end

      elif(number_of_registers == 8):
          enter_critical
              index = rq_comm_slave_id_to_index(slave_id)
              rq_comm_write_register_1000[index] = registers_100x[0]
              rq_comm_write_register_1001[index] = registers_100x[1]
              rq_comm_write_register_1002[index] = registers_100x[2]
              rq_comm_write_register_1003[index] = registers_100x[3]
              rq_comm_write_register_1004[index] = registers_100x[4]
              rq_comm_write_register_1005[index] = registers_100x[5]
              rq_comm_write_register_1006[index] = registers_100x[6]
              rq_comm_write_register_1007[index] = registers_100x[7]
              rq_comm_write_8_registers_100x_request[index] = True
          exit_critical

          while(rq_comm_write_8_registers_100x_request[index]):
              sleep(0.008)
          end

      end
  end

  def rq_comm_write_1_register_6020(slave_id, register_value):
      enter_critical
          index = rq_comm_slave_id_to_index(slave_id)
          rq_comm_write_register_6020[index] = register_value
          rq_comm_write_register_6020_request[index] = True
      exit_critical

      while(rq_comm_write_register_6020_request[index]):
          sleep(0.008)
      end
  end

  def rq_comm_get_registers_100x(slave_id, number_of_registers):
      index = rq_comm_slave_id_to_index(slave_id)

      if(number_of_registers == 3):
          return [rq_comm_write_register_1000[index],
                  rq_comm_write_register_1001[index],
                  rq_comm_write_register_1002[index]]
      elif(number_of_registers == 8):
          return [rq_comm_write_register_1000[index],
                  rq_comm_write_register_1001[index],
                  rq_comm_write_register_1002[index],
                  rq_comm_write_register_1003[index],
                  rq_comm_write_register_1004[index],
                  rq_comm_write_register_1005[index],
                  rq_comm_write_register_1006[index],
                  rq_comm_write_register_1007[index]]
      else:
          popup("Invalid number_of_registers in rq_comm_get_registers_100x(slave_id, number_of_registers)", title="rq_comm_get_registers_100x()", error=True, blocking=True)
      end
  end

  def rq_comm_read_registers_200x(slave_id, number_of_registers):
      if(number_of_registers == 3):
          enter_critical
              index = rq_comm_slave_id_to_index(slave_id)
              rq_comm_read_3_registers_200x_request[index] = True
          exit_critical

          while(rq_comm_read_3_registers_200x_request[index]):
              sleep(0.008)
          end

          return [rq_comm_read_register_2000[index],
                  rq_comm_read_register_2001[index],
                  rq_comm_read_register_2002[index]]

      elif(number_of_registers == RQ_READ_SCREWDRIVER_REGISTERS_SIZE):
          enter_critical
              index = rq_comm_slave_id_to_index(slave_id)
              rq_comm_read_22_registers_200x_request[index] = True
          exit_critical

          while(rq_comm_read_22_registers_200x_request[index]):
              sleep(0.008)
          end

          return [rq_comm_read_register_2000[index],
                  rq_comm_read_register_2001[index],
                  rq_comm_read_register_2002[index],
                  rq_comm_read_register_2003[index],
                  rq_comm_read_register_2004[index],
                  rq_comm_read_register_2005[index],
                  rq_comm_read_register_2006[index],
                  rq_comm_read_register_2007[index],
                  rq_comm_read_register_2008[index],
                  rq_comm_read_register_2009[index],
                  rq_comm_read_register_2010[index],
                  rq_comm_read_register_2011[index],
                  rq_comm_read_register_2012[index],
                  rq_comm_read_register_2013[index],
                  rq_comm_read_register_2014[index],
                  rq_comm_read_register_2015[index],
                  rq_comm_read_register_2016[index],
                  rq_comm_read_register_2017[index],
                  rq_comm_read_register_2018[index],
                  rq_comm_read_register_2019[index],
                  rq_comm_read_register_2020[index],
                  rq_comm_read_register_2021[index]]
      else:
          popup("Invalid number_of_registers in rq_comm_read_registers_200x(slave_id, number_of_registers)", title="rq_comm_read_registers_200x()", error=True, blocking=True)
      end
  end

  def rq_comm_read_registers_250x(slave_id):
      enter_critical
          index = rq_comm_slave_id_to_index(slave_id)
          rq_comm_read_registers_250x_request[index] = True
      exit_critical

      while(rq_comm_read_registers_250x_request[index]):
          sleep(0.008)
      end

      return [rq_comm_read_register_2500[index],
              rq_comm_read_register_2501[index],
              rq_comm_read_register_2502[index],
              rq_comm_read_register_2503[index],
              rq_comm_read_register_2504[index],
              rq_comm_read_register_2505[index],
              rq_comm_read_register_2506[index],
              rq_comm_read_register_2507[index],
              rq_comm_read_register_2508[index]]
  end

  def rq_comm_read_3_registers_6020(slave_id):
      enter_critical
          index = rq_comm_slave_id_to_index(slave_id)
          rq_comm_read_3_registers_602x_request[index] = True
      exit_critical

      while(rq_comm_read_3_registers_602x_request[index]):
          sleep(0.008)
      end

      return [rq_comm_read_register_6020[index],
              rq_comm_read_register_6021[index],
              rq_comm_read_register_6022[index]]
  end

  def rq_comm_slave_id_to_index(slave_id = 9):
      if(slave_id == 9):
          return 0
      else:
          return (slave_id - 1)
      end
  end

  def rq_get_number_of_slaves():
      return get_list_length(rq_comm_slave_ids)
  end

  def rq_read_registers(slave_id, start_address, number_of_registers, client_modbus):
    retries = 10
    index = rq_comm_slave_id_to_index(slave_id)
    while (retries >= 0):
      registers = client_modbus.ModbusServiceWrapper.readRegisters(slave_id, start_address, number_of_registers)

      if(get_list_length(registers) > 0):
        if(registers[0] >= 0):
          rq_comm_lost[index] = False
          break
        else:
          textmsg("An error occurred while reading modbus registers: ", rq_convert_error_number_to_exception(registers[0]))
          rq_comm_lost[index] = True
        end
      else:
        textmsg("An error occurred while reading modbus registers: ", "No registers read")
        rq_comm_lost[index] = True
      end

      retries = retries - 1
    end

    return registers
  end

  def rq_write_registers(slave_id, start_address, registers, client_modbus):
    retries = 10
    success = -1
    index = rq_comm_slave_id_to_index(slave_id)

    while (retries >= 0 and success != 0):
      success = client_modbus.ModbusServiceWrapper.writeRegisters(slave_id, start_address, registers)
      retries = retries - 1
    end
    if(success < 0):
      textmsg("An error occurred while writing modbus registers: ", rq_convert_error_number_to_exception(success))
    end

    rq_comm_lost[index] = (success < 0)

    return success
  end

  thread rq_modbus_comm():
      def rq_handle_write_requests():
          index = 0
          while(index < rq_get_number_of_slaves()):
              if(rq_comm_write_3_registers_100x_request[index]):
                  slave_id = rq_comm_slave_ids[index]
                  rq_write_registers(slave_id, 1000, rq_comm_get_registers_100x(slave_id, 3), rq_xml_rpc_modbus)
                  rq_comm_write_3_registers_100x_request[index] = False
              end
              if(rq_comm_write_8_registers_100x_request[index]):
                  slave_id = rq_comm_slave_ids[index]
                  rq_write_registers(slave_id, 1000, rq_comm_get_registers_100x(slave_id, 8),rq_xml_rpc_modbus)
                  rq_comm_write_8_registers_100x_request[index] = False
              end
              if(rq_comm_write_register_6020_request[index]):
                  slave_id = rq_comm_slave_ids[index]
                  rq_write_registers(slave_id, 6020, [rq_comm_write_register_6020[index]], rq_xml_rpc_modbus)
                  rq_comm_write_register_6020_request[index] = False
              end
              index = index + 1
          end
      end

